   // nicht in Automatik
   #Mld.n_Auto := NOT #In.Auto AND "DB_ANLAGE".BA.Automat_ein;

   // Zeitüberschreitung links öffnen
   #IEC_Timer.TO_li_auf(IN := #Out.links_auf AND NOT #In.S_links_auf,
                        PT := #Param.TO,
                        Q => #TO_links_auf);
   IF #TO_links_auf THEN
       #Mld.TO_links_auf := TRUE;
   ELSIF #In.ErrQ THEN
       #Mld.TO_links_auf := FALSE;
   END_IF;
   // Zeitüberschreitung links schließen
   #IEC_Timer.TO_li_zu(IN := #Out.links_zu AND NOT #In.S_links_zu,
                        PT := #Param.TO,
                        Q => #TO_links_zu);
    IF #TO_links_zu THEN
        #Mld.TO_links_zu := TRUE;
    ELSIF #In.ErrQ THEN
        #Mld.TO_links_zu := FALSE;
    END_IF;
     // Zeitüberschreitung rechts öffnen
    #IEC_Timer.TO_re_auf(IN := #Out.rechts_auf AND NOT #In.S_rechts_auf,
                         PT := #Param.TO,
                         Q => #TO_rechts_auf);
    IF #TO_rechts_auf THEN
        #Mld.TO_rechts_auf := TRUE;
    ELSIF #In.ErrQ THEN
        #Mld.TO_rechts_auf := FALSE;
    END_IF;
    // Zeitüberschreitung rechts schließen
    #IEC_Timer.TO_re_zu(IN := #Out.rechts_zu AND NOT #In.S_rechts_zu,
                        PT := #Param.TO,
                        Q => #TO_rechts_zu);
    IF #TO_rechts_zu THEN
        #Mld.TO_rechts_zu := TRUE;
    ELSIF #In.ErrQ THEN
        #Mld.TO_rechts_zu := FALSE;
    END_IF;
   // Sensor und SRM Zylinder Zeitfenster überwachen 
    #IEC_Timer.gleich_li_auf(IN := #In.SRM_links_auf AND NOT #In.S_links_auf,
                             PT := #Param.gleichzeitig,
                             Q => #Mld.SF_gleich_li_auf);
    // Sensor und SRM Zylinder Zeitfenster überwachen 
    #IEC_Timer.gleich_li_zu(IN := #In.SRM_links_zu AND NOT #In.S_links_zu,
                             PT := #Param.gleichzeitig,
                             Q => #Mld.SF_gleich_li_zu);
     // Sensor und SRM Zylinder Zeitfenster überwachen 
     #IEC_Timer.gleich_re_auf(IN := #In.SRM_rechts_auf AND NOT #In.S_rechts_auf,
                             PT := #Param.gleichzeitig,
                             Q => #Mld.SF_gleich_re_auf);
    // Sensor und SRM Zylinder Zeitfenster überwachen 
    #IEC_Timer.gleich_re_zu(IN := #In.SRM_rechts_zu AND NOT #In.S_rechts_zu,
                            PT := #Param.gleichzeitig,
                            Q => #Mld.SF_gleich_re_zu);
END_REGION
END_FUNCTION_BLOCK

FUNCTION_BLOCK "RT"   // FB1192, LAD
TITLE = Torsteuerung
{ S7_Optimized_Access := 'TRUE' }
// stored: AutoNumber false, MemoryReserve 100, SetENOAutomatically true
   VAR RETAIN
      In { ExternalAccessible := 'False'; ExternalVisible := 'False'; ExternalWritable := 'False'} : Struct
         NotHalt : Bool;
         MSS_ok : Bool;
         ok : Bool;
         Knauf_Auto : Bool;
         T_auf : Bool;   // Paneltaste
         T_zu : Bool;   // Paneltaste
         S_auf : Bool;
         S_zu : Bool;
         ErrQ : Bool;   // Fehlerquittung
         Sperrluft_ok : Bool;
         Kein_Gas_Alarm : Bool;
      END_STRUCT;
      Param { ExternalAccessible := 'False'; ExternalVisible := 'False'; ExternalWritable := 'False'} : Struct
         "TO" : Time := T#3s500ms;
      END_STRUCT;
      Zst { ExternalAccessible := 'False'; ExternalVisible := 'False'; ExternalWritable := 'False'} : Struct
         Req_Auf : Bool;
         Fehler : Bool;
         Sperre_QF : Bool;
         QF_sicher : Bool;
      END_STRUCT;
      Out { ExternalAccessible := 'False'; ExternalVisible := 'False'; ExternalWritable := 'False'} : Struct
         auf : Bool;
         zu : Bool;
      END_STRUCT;
      Mld { ExternalAccessible := 'False'; ExternalVisible := 'False'; ExternalWritable := 'False'} : Struct
         n_Auto : Bool;
         TO_auf : Bool;
         TO_zu : Bool;
         MSS : Bool;
         nok : Bool;
      END_STRUCT;
   END_VAR
   VAR
      IEC_Timer { ExternalAccessible := 'False'; ExternalVisible := 'False'; ExternalWritable := 'False'} : Struct
         TO_auf : TON_TIME;
         TO_zu : TON_TIME;
      END_STRUCT;
   END_VAR
   VAR_TEMP
      TO_auf : Bool;
      TO_zu : Bool;
   END_VAR
BEGIN

REGION Network 1 (SCL): Input
   // Panelbdienung und Sensoren --> Input()
   // Not-Halt
   #In.NotHalt := NOT "DB_PNOZ_IN_Out".In.NH_Frg_RT;
   // kein Gasalarm
   #In.Kein_Gas_Alarm :="E_Al_Gas_ok";
   // Sperrluftventilator an
   #In.Sperrluft_ok := "A_Frg_FU_Vent";

   // Schnittstelle zum Transportsystem
   #Zst.QF_sicher :=("E_S_Pos_BE_QF1" OR "E_S_Pos_Ue_QF1") AND ("E_S_Pos_BE_QF2" OR "E_S_Pos_Ue_QF2")
   AND NOT "A_Frg_FU_QF_WR02" AND NOT "A_Frg_FU_QF_WR03";
END_REGION

REGION Network 2 (SCL): Sammelstörung
   IF #In.ErrQ THEN
       #Zst.Fehler := FALSE;
   END_IF;
   IF #In.NotHalt OR NOT #In.MSS_ok OR NOT #In.ok OR #Mld.TO_auf OR #Mld.TO_zu THEN
       #Zst.Fehler := TRUE;
   END_IF;
END_REGION

REGION Network 3 (SCL): Ansteuerung
   IF NOT #Zst.Fehler AND #In.Kein_Gas_Alarm AND #In.Sperrluft_ok THEN
       IF #In.Knauf_Auto THEN
           // Automatikbetrieb
           IF #Zst.QF_sicher THEN
               #Out.auf := #Zst.Req_Auf;// wird von WR02/03 gebildet
               #Out.zu := NOT #Zst.Req_Auf;
           ELSE
               #Out.auf := FALSE;
               #Out.zu := FALSE;
           END_IF;
       ELSE
           // Handbetrieb
           IF #In.T_auf AND NOT #In.T_zu THEN
               #Out.auf := TRUE;
               #Out.zu := FALSE;
           END_IF;
           IF #In.T_zu AND NOT #In.T_auf AND #Zst.QF_sicher THEN
               #Out.zu := TRUE;
               #Out.auf := FALSE;
           END_IF;
       END_IF;
   ELSE // Not-Halt, n.i.O, MSS
       #Out.auf := FALSE;
       #Out.zu := FALSE;
   END_IF;

   // Endlagen erreicht
   IF #In.S_auf THEN
       #Out.auf := FALSE;
   END_IF;

   IF #In.S_zu THEN
       #Out.zu := FALSE;
   END_IF;
END_REGION

REGION Network 4 (SCL): Sperre
   // Fahrt WR02/03  verboten
   #Zst.Sperre_QF := NOT #In.S_auf OR #In.S_zu OR #Out.zu;
END_REGION

REGION Network 5 (SCL): Überwachung / Alarme
   // MSS / Zeitüberschreitung
   // nicht betriebsbereit
   #Mld.nok := NOT #In.ok AND NOT #In.NotHalt;
   // Motorschutzschalter
   #Mld.MSS := NOT #In.MSS_ok AND NOT #In.NotHalt;

   // nicht in Automatik
   #Mld.n_Auto := NOT #In.Knauf_Auto AND "DB_ANLAGE".BA.Automat_ein;

   // Zeitüberschreitung öffnen
   #IEC_Timer.TO_auf(IN := #Out.auf AND NOT #In.S_auf,
                        PT := #Param.TO,
                        Q => #TO_auf);
      IF #TO_auf THEN
          #Mld.TO_auf := TRUE;
      ELSIF #In.ErrQ THEN
          #Mld.TO_auf := FALSE;
      END_IF;
          // Zeitüberschreitung schließen
   #IEC_Timer.TO_zu(IN := #Out.zu AND NOT #In.S_zu,
                        PT := #Param.TO,
                        Q => #TO_zu);
       IF #TO_zu THEN
           #Mld.TO_zu := TRUE;
       ELSIF #In.ErrQ THEN
           #Mld.TO_zu := FALSE;
       END_IF;
END_REGION
END_FUNCTION_BLOCK

FUNCTION_BLOCK "FP_Saeure.GP0x"   // FB1001, LAD
TITLE = Filterpumpe Säure
{ S7_Optimized_Access := 'TRUE' }
// Funktionen:  Filternn / /Filterwechsel / Spülen
// stored: AutoNumber false, MemoryReserve 100, SetENOAutomatically false
   VAR RETAIN
      In { ExternalAccessible := 'False'; ExternalVisible := 'False'; ExternalWritable := 'False'} : Struct
         NotHalt : Bool;
         ext_Freigabe : Bool;   // Kein Gasalarm, Kein Notstrom
         Auto : Bool;   // Paneltaste
         Ein : Bool;   // Paneltaste
         Quitt_FW : Bool;   // Paneltaste
         FU_betriebsbereit : Bool;
         FU_Stoerung : Bool;
         Niv_TLS : Bool;
         Niv_min : Bool;
         Niv_max : Bool;
         Niv_Uel : Bool;
         Frg_Niv_CM05 : Bool;
         Leckage_ok : Bool;
         SRM_Saugseite_auf : Bool;
         SRM_Saugseite_zu : Bool;
         SRM_Eingang_Filter_auf : Bool;
         SRM_Eingang_Filter_zu : Bool;
         SRM_Ausgang_Filter_auf : Bool;
         SRM_Ausgang_Filter_zu : Bool;
         SRM_Entluften_auf : Bool;
         SRM_Entlueften_zu : Bool;
         SRM_Eingang_Spülltg_P_auf : Bool;   // Pumpe
         SRM_Eingang_Spülltg_P_zu : Bool;   // Pumpe
         SRM_Eingang_Spülltg_F_auf : Bool;   // Filter
         SRM_Eingang_Spülltg_F_zu : Bool;   // Filter
         SRM_Ausgang_Spülltg_auf : Bool;
         SRM_Ausgang_Spülltg_zu : Bool;
         Sensor_FG_links : Bool;
         Sensor_FG_rechts : Bool;
         Einhausung_HQ0x_zu : Bool;
         GW_p_FP : Bool;
         GW_p_FG : Bool;
         GW_LF_FP : Bool;
         Betriebsart : USInt := 0;   // Paneltaste
         FU_speed : Int;
         Druck_Pumpe : Real;
         Delta_p_Filter : Real;
      END_STRUCT;
      Param { ExternalAccessible := 'False'; ExternalVisible := 'False'; ExternalWritable := 'False'} : Struct
         SW_Hand : Int;   // [%]
         SW_Auto_AZ : Int;   // [%]
         SW_Auto_aAZ : Int;   // [%]
         Spülzeit_Pumpe : Time;
         FG_Zeit_leeren_Saurebecken : Time;
         FG_Zeit_leeren_CM05 : Time;
         FW_Spülzeit : Time;
         FW_Wartezeit : Time;
         FW_Zeit_fuellen : Time;
         DT_Druckaufbau : Time;
         DT_Testzeit_Pumpe : Time;
         DT_Testzeit_Filter : Time;
         SW_Drucktest_Pumpe : Real;
         SW_Drucktest_Filter : Real;
         WarnGr_FW : Real;
         Wechsel_FW : Real;
         Name_Pumpe : String[12];
         Name_Filter : String[12];
      END_STRUCT;
      Zst { ExternalAccessible := 'False'; ExternalVisible := 'False'; ExternalWritable := 'False'} : Struct
         Status_GP0x : USInt;
         Status_FW : USInt;
         Status_DT_Pumpe : USInt;
         Status_DT_Filter : USInt;
         Restzeit_Spülen_Pumpe : Time;
         Restzeit_Filter : Time;
         Restzeit_DT : Time;
         Spuelen_Pumpe : Bool;
         Spuelen_Filter : Bool;
         Spuelen_aktiv : Bool;
         Drucktest_aktiv : Bool;
         Filtern : Bool;
         Zeit_laeuft : Bool;
         Drucktest_Pu_ok : Bool;
         Drucktest_Filter_ok : Bool;
         Bedienung_erlaubt : Bool;
         speed : Int;   // [%]
      END_STRUCT;
      Mld { ExternalAccessible := 'False'; ExternalVisible := 'False'; ExternalWritable := 'False'} : Struct
         Leckage : Bool;
         GW_p_FP : Bool;
         GW_LF_FP : Bool;
         GW_p_FG : Bool;
         FG_links_nicht_zu : Bool;
         FG_rechts_nicht_zu : Bool;
         Einhausung_nicht_zu : Bool;
         FU_nicht_bereit : Bool;
         FU_Stoerung : Bool;
         FG_Spülen_Ende : Bool;
         n_Auto : Bool;
         TO_Druckaufbau : Bool;
         Drucktest_Pumpe_ok : Bool;
         Drucktest_Pumpe_Fehler : Bool;
         Pu_Spuelen_Fertig : Bool;
         Drucktest_Filter_ok : Bool;
         Drucktest_Filter_Fehler : Bool;
         Drucktest_Filter_erfordert : Bool;
         Filterbeutel_Wechsel_Vorwarngrenze : Bool;
         Filterbeutel_Wechsel_notwendig : Bool;
      END_STRUCT;
      Out { ExternalAccessible := 'False'; ExternalVisible := 'False'; ExternalWritable := 'False'} : Struct
         GP0x_Ein : Bool;
         Ventil_Saugseite : Bool;
         Ventil_Eingang_Filter : Bool;
         Ventil_Ausgang_Filter : Bool;
         Ventil_Entlueften : Bool;
         Spülventil_P_Eingang : Bool;
         Spülventil_F_Eingang : Bool;
         Spülventil_Ausgang : Bool;
         Soll_speed : Int;
      END_STRUCT;
   END_VAR
   VAR
      IEC_Timer { ExternalAccessible := 'False'; ExternalVisible := 'False'; ExternalWritable := 'False'} : Struct
         Spülen_Pumpe { S7_SetPoint := 'True'} : TP_TIME;
         Filterwechsel { S7_SetPoint := 'True'} : TP_TIME;
         GW_p { S7_SetPoint := 'True'} : TON_TIME;
         Drucktest { S7_SetPoint := 'True'} : TP_TIME;
         TO_Druckaufbau { S7_SetPoint := 'True'} : TON_TIME;
         Verz_Ueberdruck { S7_SetPoint := 'True'} : TON_TIME;
         Spülventil_Ausgang { S7_SetPoint := 'True'} : TOF_TIME;
      END_STRUCT;
      R_TRIG_Hand_EIN { ExternalAccessible := 'False'; ExternalVisible := 'False'; ExternalWritable := 'False'} : R_TRIG;
   END_VAR
   VAR_TEMP
      Spülzeit_Pumpe : Time;
      Spülzeit_Filter : Time;
      Zeit_DT : Time;
      posFl_Hand : Bool;
      Filtergehäuse_ok : Bool;
   END_VAR
   VAR CONSTANT
      Niv_TLS : USInt := 2;
      Niv_Min : USInt := 20;
      Niv_max : USInt := 90;
      Niv_Uel : USInt := 98;
      S0 : USInt := 0;
      S1 : USInt := 1;
      S2 : USInt := 2;
      S3 : USInt := 3;
      S4 : USInt := 4;
      S5 : USInt := 5;
      S6 : USInt := 6;
      S7 : USInt := 7;
      S8 : USInt := 8;
      S10_FG_Leeren : USInt := 10;
   END_VAR
BEGIN

REGION Network 1 (SCL): Input
   // Panelbedienung und Sensoren --> Input()

    // positive Flanke "Hand Ein"
   #R_TRIG_Hand_EIN(CLK := #In.Ein,
                    Q => #posFl_Hand);
END_REGION

REGION Network 2 (SCL): Ansteuerung
   // Filtergehäuse geschlossen
   #Filtergehäuse_ok := #In.Sensor_FG_links AND #In.Sensor_FG_rechts AND #In.Einhausung_HQ0x_zu;

   // Alles AUS
   IF (#In.Betriebsart = 2) AND #In.Leckage_ok AND #In.ext_Freigabe THEN // Spülen
       // Ausschaltverzögert - Druckabbau
       #IEC_Timer.Spülventil_Ausgang(IN := #Out.Spülventil_P_Eingang,
                                     PT := T#3s,
                                     Q => #Out.Spülventil_Ausgang);
   ELSE
       #Out.Spülventil_P_Eingang := FALSE;
       #Out.Spülventil_Ausgang := FALSE;
   END_IF;
   #Out.Spülventil_F_Eingang := FALSE;
   #Zst.Restzeit_Spülen_Pumpe := T#0s;
   #Zst.Restzeit_Filter := T#0s;
   #Out.Ventil_Saugseite := FALSE;
   #Out.Ventil_Eingang_Filter := FALSE;
   #Out.Ventil_Entlueften := FALSE;
   #Out.Ventil_Ausgang_Filter := FALSE;

   // "Normal"-Betrieb
   #Zst.Bedienung_erlaubt := NOT #In.Ein AND NOT #In.Auto AND NOT #Mld.Drucktest_Pumpe_Fehler AND NOT #Mld.Drucktest_Filter_Fehler;

   //Drucktest Pumpe rücksetzen
   IF #In.Betriebsart <> 3 OR #Zst.Spuelen_aktiv OR #Zst.Filtern OR NOT #In.Ein THEN
       #Mld.Drucktest_Pumpe_ok := FALSE;
       // #Mld.Drucktest_Pumpe_Fehler := FALSE;
       #Zst.Status_DT_Pumpe := 0;
       #Zst.Drucktest_aktiv := FALSE;
   END_IF;
   //Drucktest Filter rücksetzen
   IF #In.Betriebsart <> 4 OR #Zst.Spuelen_aktiv OR #Zst.Filtern OR NOT #In.Ein THEN
       #Mld.Drucktest_Filter_ok := FALSE;
       // #Mld.Drucktest_Filter_Fehler := FALSE;
       #Zst.Status_DT_Filter := 0;
   END_IF;
   IF #In.Betriebsart <> 3 AND #In.Betriebsart <> 4 THEN
       #Mld.TO_Druckaufbau := FALSE;
   END_IF;
   //Filterwechsel rücksetzen
   IF #In.Betriebsart <> 1 OR #Zst.Spuelen_aktiv OR NOT #In.Ein THEN
       #Zst.Status_FW := 0;
   END_IF;
   //Spülmeldung rücksetzen
   IF #In.Betriebsart <> 2 OR NOT #In.Ein THEN
       #Mld.Pu_Spuelen_Fertig := FALSE;
   END_IF;
   IF #In.Leckage_ok AND #In.ext_Freigabe THEN
       CASE #In.Betriebsart OF
           0:  // Filterbetrieb
                         // Ventile öffnen
               IF NOT #Mld.Drucktest_Filter_erfordert AND NOT #Mld.Filterbeutel_Wechsel_notwendig THEN
                   #Out.Ventil_Saugseite := (#In.Auto OR #In.Ein) AND #In.Niv_TLS AND #In.SRM_Ausgang_Spülltg_zu AND #In.SRM_Eingang_Spülltg_P_zu AND #In.SRM_Eingang_Spülltg_F_zu;
                   #Out.Ventil_Eingang_Filter := #Out.Ventil_Saugseite;
                   #Out.Ventil_Ausgang_Filter := #Out.Ventil_Eingang_Filter;
               END_IF;
                   // Wenn geöffnet --> Frg Pumpe
                   #Zst.Filtern := #In.SRM_Eingang_Filter_auf AND #In.SRM_Ausgang_Filter_auf AND #In.SRM_Saugseite_auf;
                   // #Zst.Status_FW := #Ende;

           1:  // Filterwechsel 
               REGION Filterwechsel
                   #Zst.Filtern := FALSE;
                   CASE #Zst.Status_FW OF
                       #S0:  // Grundzustand
                           IF #In.Auto OR #In.Ein THEN
                               #Zst.Status_FW := #S1;
                           END_IF;

                       #S1:    // 1. Mal Leerlaufen ins Säurebecken - vor Spülen: Pumpe Aus - Ventile Auf - Zeit warten
                           // Ventile öffnen
                           #Out.Ventil_Eingang_Filter := #Filtergehäuse_ok AND #In.SRM_Ausgang_Spülltg_zu AND #In.SRM_Eingang_Spülltg_P_zu AND #In.SRM_Eingang_Spülltg_F_zu;
                           #Out.Ventil_Ausgang_Filter := #Out.Ventil_Eingang_Filter;
                           #Out.Ventil_Saugseite := #Out.Ventil_Eingang_Filter;
                           #Out.Ventil_Entlueften := #Out.Ventil_Eingang_Filter;

                           #IEC_Timer.Filterwechsel(IN := #In.SRM_Eingang_Filter_auf AND #In.SRM_Ausgang_Filter_auf AND #In.SRM_Saugseite_auf AND #In.SRM_Entluften_auf,
                                                    PT := #Param.FG_Zeit_leeren_Saurebecken,
                                                    ET => #Spülzeit_Filter,
                                                    Q => #Zst.Zeit_laeuft);
                           #Zst.Restzeit_Filter := #Param.FG_Zeit_leeren_Saurebecken - #Spülzeit_Filter;

                           IF NOT #Zst.Zeit_laeuft AND #In.SRM_Eingang_Filter_auf AND #In.SRM_Ausgang_Filter_auf AND #In.SRM_Saugseite_auf AND #In.SRM_Entluften_auf THEN
                               #Out.Ventil_Ausgang_Filter := #Out.Ventil_Eingang_Filter := #Out.Ventil_Saugseite := #Out.Ventil_Entlueften := FALSE;
                               #Zst.Status_FW := #S2;
                           END_IF;

                       #S2:    // Spülen Filtergehäuse
                           // Ventile öffnen
                           #Out.Spülventil_F_Eingang := #In.Frg_Niv_CM05;
                           #Out.Spülventil_Ausgang := NOT #Out.Ventil_Entlueften;
                           #Out.Ventil_Entlueften := #Zst.Zeit_laeuft AND #Zst.Restzeit_Filter < T#15s; //#Spülzeit_Filter > T#45s AND #Spülzeit_Filter <= T#60s;
                           #IEC_Timer.Filterwechsel(IN := #In.SRM_Ausgang_Spülltg_auf AND #In.SRM_Eingang_Spülltg_F_auf,
                                                    PT := #Param.FW_Spülzeit,
                                                    ET => #Spülzeit_Filter,
                                                    Q => #Zst.Zeit_laeuft);
                           #Zst.Restzeit_Filter := #Param.FW_Spülzeit - #Spülzeit_Filter;

                           IF NOT #Zst.Zeit_laeuft AND #In.SRM_Ausgang_Spülltg_auf AND #In.SRM_Eingang_Spülltg_F_auf THEN
                               #Out.Spülventil_F_Eingang := #Out.Spülventil_Ausgang := FALSE;
                               #Out.Ventil_Entlueften := FALSE;
                               #Zst.Status_FW := #S3;
                           END_IF;

                       #S3:    // Warten --> Meldung
                           #IEC_Timer.Filterwechsel(IN := #In.SRM_Ausgang_Spülltg_zu AND #In.SRM_Eingang_Spülltg_F_zu AND #In.SRM_Entlueften_zu,
                                                    PT := #Param.FW_Wartezeit,
                                                    ET => #Spülzeit_Filter,
                                                    Q => #Zst.Zeit_laeuft);
                           #Zst.Restzeit_Filter := #Param.FW_Wartezeit - #Spülzeit_Filter;
                           // Ventile öffnen
                           IF #Zst.Zeit_laeuft AND #Zst.Restzeit_Filter < t#10s THEN
                               #Out.Ventil_Entlueften := TRUE;// #Zst.Zeit_laeuft AND #Zst.Restzeit_Filter < t#10s; // #Spülzeit_Filter > T#45s AND #Spülzeit_Filter <= T#60s;
                               #Out.Spülventil_F_Eingang := #Out.Ventil_Entlueften;
                           ELSE
                               #Out.Ventil_Entlueften := FALSE;
                               #Out.Spülventil_F_Eingang := FALSE;
                           END_IF;

                           IF NOT #Zst.Zeit_laeuft AND #In.SRM_Eingang_Spülltg_F_auf AND #In.SRM_Entluften_auf THEN
                               #Zst.Status_FW := #S4;
                           END_IF;

                       #S4:    // 2. Mal Leerlaufen in CM05 - nach Spülen: Pumpe Aus - Ventile Auf - Zeit warten
                           // Ventile öffnen
                           #Out.Ventil_Saugseite := FALSE;
                         //  #Out.Ventil_Eingang_Filter := FALSE;  04.08.21
                           #Out.Spülventil_Ausgang :=  #In.Frg_Niv_CM05 (*AND #In.SRM_Ausgang_Filter_zu 04.08.21*) AND #In.SRM_Eingang_Spülltg_P_zu AND #In.SRM_Eingang_Spülltg_F_zu;
                           #Out.Ventil_Entlueften := #Out.Spülventil_Ausgang;

                           #IEC_Timer.Filterwechsel(IN :=  #In.Frg_Niv_CM05 (*AND #In.SRM_Eingang_Filter_zu 04.08.21*) AND #In.SRM_Ausgang_Spülltg_auf AND #In.SRM_Saugseite_zu AND #In.SRM_Entluften_auf,
                                                    PT := #Param.FG_Zeit_leeren_CM05,
                                                    ET => #Spülzeit_Filter,
                                                    Q => #Zst.Zeit_laeuft);
                           #Zst.Restzeit_Filter := #Param.FG_Zeit_leeren_CM05 - #Spülzeit_Filter;

                           // 03.08.21
                           //Eine Bitte habe ich noch, zwar beim Filterwechsel. Es steht immer noch recht viel restliches saures Wasser im Behälter,
                           //könntest du bitte für den letzten Schritt noch 10sec für HQ01 den QM23 und bei HQ02 den QM60 öffnen.
                           //Somit ist auch die Leitung zur Leitfähigkeitsmessung leer.
                           #Out.Ventil_Eingang_Filter := #Out.Ventil_Ausgang_Filter := #Zst.Zeit_laeuft AND #Zst.Restzeit_Filter <= t#40s;// 03.08.21

                           IF NOT #Zst.Zeit_laeuft (*AND #In.SRM_Eingang_Filter_zu 04.08.21*) AND #In.SRM_Ausgang_Spülltg_auf AND #In.SRM_Saugseite_zu AND #In.SRM_Entluften_auf THEN
                               #Out.Ventil_Ausgang_Filter := #Out.Ventil_Eingang_Filter := #Out.Ventil_Saugseite := #Out.Ventil_Entlueften := FALSE;
                               #Zst.Status_FW := #S5;
                               #Mld.FG_Spülen_Ende := TRUE;
                           END_IF;

                       #S5:    // man.Wechsel --> Quittierung
                           // Ventile bleiben offen --> Nachlauf Restwasser in CM05
                           #Out.Ventil_Saugseite := FALSE;
                           #Out.Ventil_Eingang_Filter := FALSE;
                           #Out.Spülventil_Ausgang := #In.Frg_Niv_CM05 AND #In.SRM_Ausgang_Filter_zu AND #In.SRM_Eingang_Spülltg_P_zu AND #In.SRM_Eingang_Spülltg_F_zu;
                           #Out.Ventil_Entlueften := #Out.Spülventil_Ausgang;

                           IF #Filtergehäuse_ok AND #In.Quitt_FW THEN
                               #Mld.FG_Spülen_Ende := FALSE;
                               #Mld.Drucktest_Filter_erfordert := TRUE;
                               #Mld.Filterbeutel_Wechsel_notwendig := FALSE;
                               #In.Quitt_FW := FALSE;
                               #Zst.Status_FW := #S8;
                           END_IF;

                           (*     
                            #S6:    //Filtergehäuse füllen
                                #Out.Ventil_Saugseite := (#In.Auto OR #In.Ein) AND #In.Niv_TLS AND #In.SRM_Ausgang_Spülltg_zu AND #In.SRM_Eingang_Spülltg_P_zu AND #In.SRM_Eingang_Spülltg_F_zu;
                                #Out.Ventil_Eingang_Filter := #Out.Ventil_Saugseite;
                                #Out.Ventil_Ausgang_Filter := TRUE;
                                #Out.Spülventil_Ausgang := FALSE;

                                // Wenn geöffnet --> Frg Pumpe
                                #IEC_Timer.Filterwechsel(IN := #In.SRM_Eingang_Filter_auf AND #In.SRM_Saugseite_auf AND #In.SRM_Ausgang_Filter_auf,
                                                         PT := #Param.FW_Zeit_fuellen,
                                                         ET => #Spülzeit_Filter,
                                                         Q => #Zst.Zeit_laeuft);

                                #Zst.Filtern := #In.SRM_Eingang_Filter_auf AND #In.SRM_Ausgang_Filter_auf AND #In.SRM_Saugseite_auf;

                                #Zst.Restzeit_Filter := #Param.FW_Zeit_fuellen - #Spülzeit_Filter;

                                IF NOT #Zst.Zeit_laeuft AND #Zst.Filtern THEN
                                    #Zst.Status_FW := #S7;
                                END_IF;


                            #S7:    // Kreislauf öffnen
                                // #Out.Ventil_Ausgang_Filter := TRUE;
                                // #Out.Spülventil_Ausgang := NOT #In.SRM_Ausgang_Filter_auf;

                                // IF #In.SRM_Ausgang_Filter_auf AND #In.SRM_Ausgang_Spülltg_zu THEN
                                //     #Zst.Status_FW := #S8;
                                // END_IF;
                                #Zst.Filtern := FALSE;
                                IF #Zst.speed <= 20 THEN
                                    #Out.Ventil_Saugseite := FALSE;
                                    #Out.Ventil_Eingang_Filter := FALSE;
                                    #Out.Ventil_Ausgang_Filter := FALSE;
                                    #Out.Spülventil_Ausgang := FALSE;
                                END_IF;

                                IF NOT  #Zst.Filtern AND  #In.SRM_Saugseite_zu AND #In.SRM_Eingang_Filter_zu AND #In.SRM_Ausgang_Filter_zu AND #In.SRM_Ausgang_Spülltg_zu THEN
                                    #Zst.Status_FW := #S8;
                                END_IF;
                                  *)
                       #S8: // Ende
                           ;
                   END_CASE;
               END_REGION

           2:// Spülen - nur Hand
               #Zst.Filtern := FALSE;
               #Zst.Status_FW := #S0;

               IF NOT #Mld.Drucktest_Filter_erfordert AND NOT #Mld.Filterbeutel_Wechsel_notwendig THEN
                   IF #In.Ein AND #In.Frg_Niv_CM05 THEN
                       IF #posFl_Hand THEN
                           #Zst.Spuelen_aktiv := TRUE;
                       END_IF;
                       #Out.Spülventil_P_Eingang := #Filtergehäuse_ok AND #In.SRM_Ausgang_Filter_zu AND #In.SRM_Saugseite_zu AND #Zst.Spuelen_aktiv;
                       #Out.Ventil_Eingang_Filter := #Out.Spülventil_Ausgang;

                       #IEC_Timer.Spülen_Pumpe(IN := #In.SRM_Eingang_Spülltg_P_auf AND #In.SRM_Ausgang_Spülltg_auf,
                                               PT := #Param.Spülzeit_Pumpe,
                                               Q => #Zst.Spuelen_Pumpe,
                                               ET => #Spülzeit_Pumpe);
                       #Zst.Restzeit_Spülen_Pumpe := #Param.Spülzeit_Pumpe - #Spülzeit_Pumpe;

                       IF #In.SRM_Eingang_Spülltg_P_auf AND #In.SRM_Ausgang_Spülltg_auf AND NOT #Zst.Spuelen_Pumpe THEN
                           #Zst.Spuelen_aktiv := FALSE;
                           #Out.Spülventil_P_Eingang := FALSE;
                       END_IF;

                       // Fertig
                       IF NOT #Zst.Spuelen_Pumpe AND NOT #Zst.Spuelen_aktiv AND NOT #Out.Spülventil_Ausgang THEN
                           #Out.Spülventil_P_Eingang := FALSE;
                           #Out.Spülventil_Ausgang := FALSE;
                           #Out.Ventil_Eingang_Filter := FALSE;
                           #Zst.Restzeit_Spülen_Pumpe := T#0s;
                           #Mld.Pu_Spuelen_Fertig := TRUE;
                       END_IF;
                   ELSE
                       #Zst.Spuelen_Pumpe := FALSE;
                       #Out.Spülventil_P_Eingang := FALSE;
                       #Out.Spülventil_Ausgang := FALSE;
                       #Out.Ventil_Eingang_Filter := FALSE;
                       #Zst.Restzeit_Spülen_Pumpe := T#0s;
                   END_IF;
                   // Ausschaltverzögert - Druckabbau
                   #IEC_Timer.Spülventil_Ausgang(IN := #Out.Spülventil_P_Eingang,
                                                 PT := T#3s,
                                                 Q => #Out.Spülventil_Ausgang);
               END_IF;
           3: // Spülen + Drucktest - nur Hand
               #Zst.Filtern := FALSE;
               #Zst.Status_FW := #S0;
               IF NOT #Mld.Drucktest_Filter_erfordert AND NOT #Mld.Filterbeutel_Wechsel_notwendig THEN
                   IF NOT #Zst.Drucktest_aktiv THEN
                       IF #In.Ein AND #In.Frg_Niv_CM05 THEN
                           IF #posFl_Hand THEN
                               #Zst.Spuelen_aktiv := TRUE;
                           END_IF;
                           #Out.Spülventil_P_Eingang := #Filtergehäuse_ok AND #In.SRM_Ausgang_Filter_zu AND #In.SRM_Saugseite_zu;
                           #Out.Spülventil_Ausgang := #Out.Spülventil_P_Eingang;
                           #Out.Ventil_Eingang_Filter := #Out.Spülventil_P_Eingang;

                           #IEC_Timer.Spülen_Pumpe(IN := #In.SRM_Eingang_Spülltg_P_auf AND #In.SRM_Ausgang_Spülltg_auf,
                                                   PT := #Param.Spülzeit_Pumpe,
                                                   Q => #Zst.Spuelen_Pumpe,
                                                   ET => #Spülzeit_Pumpe);
                           #Zst.Restzeit_Spülen_Pumpe := #Param.Spülzeit_Pumpe - #Spülzeit_Pumpe;

                           IF #In.SRM_Eingang_Spülltg_P_auf AND #In.SRM_Ausgang_Spülltg_auf AND NOT #Zst.Spuelen_Pumpe THEN
                               #Zst.Spuelen_aktiv := FALSE;
                           END_IF;

                           // Fertig
                           IF NOT #Zst.Spuelen_Pumpe AND NOT #Zst.Spuelen_aktiv THEN
                               #Out.Spülventil_Ausgang := FALSE;
                               #Out.Ventil_Eingang_Filter := FALSE;
                               #Zst.Restzeit_Spülen_Pumpe := T#0s;
                               #Zst.Drucktest_aktiv := TRUE;
                               #Zst.Status_DT_Pumpe := #S1;
                           END_IF;
                       ELSE
                           #Zst.Spuelen_Pumpe := FALSE;
                           #Out.Spülventil_P_Eingang := FALSE;
                           #Out.Spülventil_Ausgang := FALSE;
                           #Out.Ventil_Eingang_Filter := FALSE;
                           #Zst.Restzeit_Spülen_Pumpe := T#0s;
                       END_IF;
                   END_IF;


                   //Drucktest
                   IF #Zst.Drucktest_aktiv THEN

                       CASE #Zst.Status_DT_Pumpe OF
                           #S1:  //Druckaufbau

                               IF "DB_Temporaer".Drucksensoren_deaktiviert THEN //20.01.22
                                   #Zst.Drucktest_Pu_ok := TRUE;

                                   "Ergebnis_DT"("Name" := #Param.Name_Pumpe,
                                                 akt_Zeit := "Uhrzeit".aktDatum,
                                                 ok := #Zst.Drucktest_Pu_ok,
                                                 Fehler := NOT #Zst.Drucktest_Pu_ok);

                                   #Mld.Drucktest_Pumpe_ok := #Zst.Drucktest_Pu_ok;
                                   #Mld.Drucktest_Pumpe_Fehler := NOT #Zst.Drucktest_Pu_ok;

                                   #Zst.Status_DT_Pumpe := #S4;
                               ELSE
                                   #Out.Spülventil_P_Eingang := #In.SRM_Ausgang_Filter_zu AND #In.SRM_Saugseite_zu;
                                   #Out.Ventil_Eingang_Filter := FALSE;
                                   #Out.Spülventil_Ausgang := FALSE;

                                   IF (#In.Druck_Pumpe > #Param.SW_Drucktest_Pumpe + 0.25 AND #In.SRM_Eingang_Filter_zu) OR #Mld.TO_Druckaufbau THEN
                                       #Out.Spülventil_P_Eingang := FALSE;
                                       #Zst.Status_DT_Pumpe := #S2;
                                   END_IF;

                               END_IF;

                           #S2: //Wartezeit
                               #IEC_Timer.Drucktest(IN := #In.SRM_Eingang_Spülltg_P_zu,
                                                    PT := #Param.DT_Testzeit_Pumpe,
                                                    Q => #Zst.Zeit_laeuft,
                                                    ET => #Zeit_DT);
                               #Zst.Restzeit_DT := #Param.DT_Testzeit_Pumpe - #Zeit_DT;

                               IF NOT #Zst.Zeit_laeuft AND #In.SRM_Eingang_Spülltg_P_zu THEN
                                   #Zst.Restzeit_DT := T#0s;
                                   #Zst.Status_DT_Pumpe := #S3;
                               END_IF;

                           #S3:// Überprüfung
                               #Zst.Drucktest_Pu_ok := #In.Druck_Pumpe >= #Param.SW_Drucktest_Pumpe;

                               "Ergebnis_DT"("Name" := #Param.Name_Pumpe,
                                             akt_Zeit := "Uhrzeit".aktDatum,
                                             ok := #Zst.Drucktest_Pu_ok,
                                             Fehler := NOT #Zst.Drucktest_Pu_ok);

                               #Mld.Drucktest_Pumpe_ok := #Zst.Drucktest_Pu_ok;
                               #Mld.Drucktest_Pumpe_Fehler := NOT #Zst.Drucktest_Pu_ok;

                               #Zst.Status_DT_Pumpe := #S4;

                           #S4: // ENDE
                               ;
                       END_CASE;
                   END_IF;
               END_IF;
           4: // Drucktest Filter
               #Zst.Filtern := FALSE;
               IF #posFl_Hand (*AND NOT #Mld.Filterbeutel_Wechsel_notwendig - 23.08.22, falls während Drucktest die Meldung aktiv wird, dass es nicht im deadlock ist*) THEN
                   #Zst.Status_DT_Filter:= 1;
               END_IF;

               CASE #Zst.Status_DT_Filter OF
                   #S1:  //Druckaufbau

                       IF "DB_Temporaer".Drucksensoren_deaktiviert THEN //20.01.22
                           #Zst.Drucktest_Filter_ok := TRUE;

                           "Ergebnis_DT"("Name" := #Param.Name_Filter,
                                         akt_Zeit := "Uhrzeit".aktDatum,
                                         ok := #Zst.Drucktest_Filter_ok,
                                         Fehler := NOT #Zst.Drucktest_Filter_ok);

                           #Mld.Drucktest_Filter_ok := #Zst.Drucktest_Filter_ok;
                           #Mld.Drucktest_Filter_Fehler := NOT #Zst.Drucktest_Filter_ok;
                           #Mld.Drucktest_Filter_erfordert := FALSE;
                           #Zst.Status_DT_Filter := #S10_FG_Leeren;

                       ELSE
                           #Out.Spülventil_F_Eingang := #Filtergehäuse_ok AND #In.SRM_Ausgang_Filter_zu AND #In.SRM_Saugseite_zu;
                           #Out.Ventil_Eingang_Filter := FALSE;
                           #Out.Spülventil_Ausgang := FALSE;

                           IF (ABS(#In.Delta_p_Filter) > #Param.SW_Drucktest_Filter + 0.25 AND #In.SRM_Eingang_Spülltg_F_auf) OR #Mld.TO_Druckaufbau OR #Mld.GW_p_FG THEN
                               #Out.Spülventil_F_Eingang := FALSE;
                               #Zst.Status_DT_Filter := #S2;
                           END_IF;
                           #Zst.Restzeit_DT := #Param.DT_Druckaufbau - #IEC_Timer.TO_Druckaufbau.ET;

                       END_IF;

                   #S2: //Wartezeit
                       #IEC_Timer.Drucktest(IN := #In.SRM_Eingang_Spülltg_F_zu,
                                            PT := #Param.DT_Testzeit_Filter,
                                            Q => #Zst.Zeit_laeuft,
                                            ET => #Zeit_DT);
                       #Zst.Restzeit_DT := #Param.DT_Testzeit_Filter - #Zeit_DT;

                       IF NOT #Zst.Zeit_laeuft AND #In.SRM_Eingang_Spülltg_F_zu THEN
                           #Zst.Restzeit_DT := T#0s;
                           #Zst.Status_DT_Filter := #S3;
                       END_IF;

                   #S3:// Überprüfung
                       #Zst.Drucktest_Filter_ok := ABS(#In.Delta_p_Filter) >= #Param.SW_Drucktest_Filter;

                       "Ergebnis_DT"("Name" := #Param.Name_Filter,
                                     akt_Zeit := "Uhrzeit".aktDatum,
                                     ok := #Zst.Drucktest_Filter_ok,
                                     Fehler := NOT #Zst.Drucktest_Filter_ok);

                       #Mld.Drucktest_Filter_ok := #Zst.Drucktest_Filter_ok;
                       #Mld.Drucktest_Filter_Fehler := NOT #Zst.Drucktest_Filter_ok;
                       #Mld.Drucktest_Filter_erfordert := FALSE;
                       #Zst.Status_DT_Filter := #S10_FG_Leeren;

                   #S10_FG_Leeren: // Filtergehäuse nach NIO Drucktest leeren in CM05
                       // Ventile öffnen
                       #Out.Ventil_Saugseite := FALSE;
                     //#Out.Ventil_Eingang_Filter := FALSE;  04.08.21
                       #Out.Spülventil_Ausgang := #In.Frg_Niv_CM05 (*AND #In.SRM_Ausgang_Filter_zu 04.08.21*) AND #In.SRM_Eingang_Spülltg_P_zu AND #In.SRM_Eingang_Spülltg_F_zu;;
                       #Out.Ventil_Entlueften :=  #Out.Spülventil_Ausgang;

                       #IEC_Timer.Filterwechsel(IN := #In.Frg_Niv_CM05 (*AND #In.SRM_Eingang_Filter_zu04.08.21*)AND #In.SRM_Ausgang_Spülltg_auf AND #In.SRM_Saugseite_zu AND #In.SRM_Entluften_auf,
                                                PT := #Param.FG_Zeit_leeren_CM05,
                                                ET => #Spülzeit_Filter,
                                                Q => #Zst.Zeit_laeuft);
                       #Zst.Restzeit_DT := #Param.FG_Zeit_leeren_CM05 - #Spülzeit_Filter;

                       // 04.08.21
                       //Eine Bitte habe ich noch, zwar beim Filterwechsel. Es steht immer noch recht viel restliches saures Wasser im Behälter,
                       //könntest du bitte für den letzten Schritt noch 10sec für HQ01 den QM23 und bei HQ02 den QM60 öffnen.
                       //Somit ist auch die Leitung zur Leitfähigkeitsmessung leer.
                       #Out.Ventil_Eingang_Filter := #Out.Ventil_Ausgang_Filter := #Zst.Zeit_laeuft AND #Zst.Restzeit_DT <= t#40s;// 03.08.21

                       IF NOT #Zst.Zeit_laeuft (*AND #In.SRM_Eingang_Filter_zu04.08.21*)AND #In.SRM_Ausgang_Spülltg_auf AND #In.SRM_Saugseite_zu AND #In.SRM_Entluften_auf THEN
                           #Out.Spülventil_Ausgang := #Out.Ventil_Eingang_Filter := #Out.Ventil_Saugseite := #Out.Ventil_Entlueften := FALSE;
                           #Zst.Status_DT_Filter := #S4;
                       END_IF;

                   #S4: // ENDE
                       ;


               END_CASE;

       END_CASE;
   END_IF;

       // Pumpe an    
   #Out.GP0x_Ein := #Zst.Filtern AND NOT #In.NotHalt AND #Filtergehäuse_ok AND #In.Leckage_ok AND #In.ext_Freigabe AND (#In.Ein OR #In.Auto);

       // Geschwindigkeitsvorgabe
       // SEW: 100% == 3000 U/min == 15000 Digits
       IF #Out.GP0x_Ein THEN
           IF #In.Ein THEN
               #Out.Soll_speed := #Param.SW_Hand * 150;
           ELSE
               IF "Uhrzeit".AZ_aktiv THEN
                   #Out.Soll_speed := #Param.SW_Auto_AZ * 150;
               ELSE
                   #Out.Soll_speed := #Param.SW_Auto_aAZ * 150;
               END_IF;
           END_IF;
       ELSE
           #Out.Soll_speed := 0;
       END_IF;
END_REGION

REGION Network 3 (SCL): Überwachung / Meldungen
   // Leckage
   #Mld.Leckage := NOT #In.Leckage_ok;

   // Zeitüberschreitung Druckaufbau
   #IEC_Timer.TO_Druckaufbau(IN := #Zst.Status_DT_Pumpe = #S1 OR #Zst.Status_DT_Filter = #S1,
                             PT := #Param.DT_Druckaufbau,
                             Q => #Mld.TO_Druckaufbau);

   //Grenzwert Druck Filtergehäuse
   #IEC_Timer.Verz_Ueberdruck(IN := #In.GW_p_FG,
                              PT :=t#3s,
                              Q => #Mld.GW_p_FG);

   // Nicht geschlossen
   #Mld.Einhausung_nicht_zu := NOT #In.Einhausung_HQ0x_zu;
   #Mld.FG_links_nicht_zu := NOT #In.Sensor_FG_links;
   #Mld.FG_rechts_nicht_zu := NOT #In.Sensor_FG_rechts;

   // Grenzwert Druck Pumpe
   #IEC_Timer.GW_p(IN :=#Out.GP0x_Ein AND #In.GW_p_FP,
                   PT := T#3s,
                   Q => #Mld.GW_p_FP);
   // Grenzwert Leitfähigkeit
   #Mld.GW_LF_FP := #In.GW_LF_FP;

   // Frequenzumrichter 24V-Betrieb
   #Mld.FU_nicht_bereit := NOT #In.FU_betriebsbereit AND NOT #In.NotHalt;
   // Störung Frequenzumrichter
   #Mld.FU_Stoerung := #In.FU_Stoerung AND NOT #In.NotHalt;
   // nicht in Automatik
   #Mld.n_Auto := NOT #In.Auto AND "DB_ANLAGE".BA.Automat_ein;
   // Filterwechsel
   #Mld.Filterbeutel_Wechsel_Vorwarngrenze := #In.Delta_p_Filter > #Param.WarnGr_FW AND NOT #Mld.Filterbeutel_Wechsel_notwendig;

   IF #In.Delta_p_Filter > #Param.Wechsel_FW THEN
       #Mld.Filterbeutel_Wechsel_notwendig := TRUE;
   END_IF;
END_REGION

REGION Network 4 (SCL): --> Visu
   // Status Pumpe
   "Status_E0A"(Hand := #In.Ein,
                Auto := #In.Auto,
                SonderModus_PumpeSpuelen:=#Zst.Spuelen_Pumpe,
                Stoerung := #In.FU_Stoerung OR NOT #In.FU_betriebsbereit,
                Ausgang := #Out.GP0x_Ein,
                StatusByte => #Zst.Status_GP0x);

   // Ist-Geschwindigkeit FU
   // SEW: 100% == 3000 U/min == 15000 Digits
   #Zst.speed := #In.FU_speed / 150; // in[%]
END_REGION
END_FUNCTION_BLOCK

FUNCTION_BLOCK "UP_Saeure.GP0x"   // FB1002, LAD
TITLE = Pumpe Umwälzpumpe Säure
{ S7_Optimized_Access := 'TRUE' }
// Funktionen: Umwälzen / Entsorgung
// stored: AutoNumber false, MemoryReserve 100, SetENOAutomatically false
   VAR RETAIN
      In { ExternalAccessible := 'False'; ExternalVisible := 'False'; ExternalWritable := 'False'} : Struct
         NotHalt : Bool;
         ext_Freigabe : Bool;   // Kein Gasalarm, Kein Notstrom
         TW_senkt : Bool;
         Auto : Bool;   // Paneltaste
         Ein : Bool;   // Paneltaste
         Quitt_Al_Dfl : Bool;
         FU_betriebsbereit : Bool;
         FU_Stoerung : Bool;
         Niv_TLS : Bool;
         Niv_min : Bool;
         Niv_max : Bool;
         Niv_Uel : Bool;
         Frg_Niv_CM05 : Bool;
         SRM_Saugseite_auf : Bool;
         SRM_Saugseite_zu : Bool;
         SRM_Druckseite_auf : Bool;
         SRM_Druckseite_zu : Bool;
         SRM_Eingang_Spülltg_auf : Bool;
         SRM_Eingang_Spülltg_zu : Bool;
         SRM_Ausgang_Spülltg_auf : Bool;
         SRM_Ausgang_Spülltg_zu : Bool;
         SRM_Entsogung_UV02_auf : Bool;
         SRM_Entsogung_UV02_zu : Bool;
         SRM_UV02_GP01_auf : Bool;
         SRM_UV02_GP01_zu : Bool;
         SRM_UV02_GP02_auf : Bool;
         SRM_UV02_GP02_zu : Bool;
         "SRM_GP02.QM41_auf" : Bool;
         "SRM_GP01.QM14_auf" : Bool;
         Anf_HF_Ents_CM0x : Bool;
         GW_p_UP : Bool;
         GW_LF_UP : Bool;
         Imp_Dfl : Bool;
         GW_Dfl : Bool;
         Tuer_zu_Seite_GP01 : Bool;
         Tuer_zu_vorn_GP01 : Bool;
         Tuer_zu_vorn_GP02 : Bool;
         Leckage_Doppelrohr_ok_BL26 : Bool;
         Leckage_Doppelschlauch_ok_BL33 : Bool;
         Leckage_Uml_Tunnel_ok_BL34 : Bool;
         Leckage_PFA_Uebergang_ok_BL16 : Bool;
         Leckage_PFA_Uebergang_ok_BL25 : Bool;
         Betriebsart : USInt := 0;   // Paneltaste
         FU_speed : Int;
         Druck_Pumpe : Real;
      END_STRUCT;
      Param { ExternalAccessible := 'False'; ExternalVisible := 'False'; ExternalWritable := 'False'} : Struct
         SW_Hand : Int;   // [%]
         SW_Auto_AZ : Int;   // [%]
         SW_Auto_aAZ : Int;   // [%]
         Spülzeit : Time;
         DT_Druckaufbau : Time;
         DT_Testzeit : Time;
         SW_Drucktest : Real;
         "Name" : String[12];
      END_STRUCT;
      Zst { ExternalAccessible := 'False'; ExternalVisible := 'False'; ExternalWritable := 'False'} : Struct
         Niveau : USInt;
         Status_GP0x : USInt;
         Status_DT : USInt;
         Restzeit_Spülen : Time;
         Restzeit_DT : Time;
         Spuelen : Bool;
         Spuelen_aktiv : Bool;
         Drucktest_aktiv : Bool;
         Umwaelzen : Bool;
         Weg_frei : Bool;
         Zeit_laeuft : Bool;
         Drucktest_ok : Bool;
         Bedienung_erlaubt : Bool;
         speed : Int;   // [%]
      END_STRUCT;
      Mld { ExternalAccessible := 'False'; ExternalVisible := 'False'; ExternalWritable := 'False'} : Struct
         Niv_TLS : Bool;
         Niv_Ueberlauf : Bool;
         Niv_Sensorfehler : Bool;
         GW_p_UP : Bool;
         GW_LF_UP : Bool;
         GW_Dfl : Bool;
         UeW_Dfl_Ents : Bool;
         FU_nicht_bereit : Bool;
         FU_Stoerung : Bool;
         n_Auto : Bool;
         TO_Druckaufbau : Bool;
         Drucktest_ok : Bool;
         DT_Fehler : Bool;
         Pu_Spuelen_Fertig : Bool;
      END_STRUCT;
      Out { ExternalAccessible := 'False'; ExternalVisible := 'False'; ExternalWritable := 'False'} : Struct
         GP0x_Ein : Bool;
         Ventil_Saugseite : Bool;
         Ventil_Druckseite : Bool;
         Spülventil_Eingang : Bool;
         Spülventil_Ausgang : Bool;
         Entsorgung_UV02 : Bool;
         Ventil_UV02_GP01 : Bool;
         Ventil_UV02_GP02 : Bool;
         Soll_speed : Int;
      END_STRUCT;
   END_VAR
   VAR
      IEC_Timer { ExternalAccessible := 'False'; ExternalVisible := 'False'; ExternalWritable := 'False'} : Struct
         Spülen { S7_SetPoint := 'True'} : TP_TIME;
         GW_p { S7_SetPoint := 'True'} : TON_TIME;
         GW_Dfl { S7_SetPoint := 'True'} : TON_TIME;
         Imp_Dfl { S7_SetPoint := 'True'} : TON_TIME;
         Drucktest { S7_SetPoint := 'True'} : TP_TIME;
         TO_Druckaufbau { S7_SetPoint := 'True'} : TON_TIME;
         Spülventil_Ausgang { S7_SetPoint := 'True'} : TOF_TIME;
      END_STRUCT;
      R_TRIG_Hand_EIN { ExternalAccessible := 'False'; ExternalVisible := 'False'; ExternalWritable := 'False'} : R_TRIG;
   END_VAR
   VAR_TEMP
      Spülzeit : Time;
      Zeit_DT : Time;
      posFl_Hand : Bool;
      Leckage_Entsorgung_ok_GP01 : Bool;
      Leckage_Entsorgung_ok_GP02 : Bool;
      Alarm_Dfl_Ents : Bool;
   END_VAR
   VAR CONSTANT
      Niv_TLS : USInt := 7;
      Niv_Min : USInt := 70;
      Niv_max : USInt := 85;
      Niv_Uel : USInt := 98;
      S1 : USInt := 1;
      S2 : USInt := 2;
      S3 : USInt := 3;
      S4 : USInt := 4;
   END_VAR
BEGIN

REGION Network 1 (SCL): Input
   // Panelbedienung und Sensoren --> Input()
   // Not-Halt
   #In.NotHalt := NOT "DB_PNOZ_IN_Out".In.NH_Frg_Pumpen OR NOT "E_Frg_AbLW";

    // positive Flanke "Hand Ein"
   #R_TRIG_Hand_EIN(CLK := #In.Ein,
                    Q => #posFl_Hand);

   // Leckage Entsorgung
   #Leckage_Entsorgung_ok_GP01 :=#In.Leckage_PFA_Uebergang_ok_BL16 AND #In.Leckage_Doppelrohr_ok_BL26 AND #In.Leckage_Uml_Tunnel_ok_BL34;

   #Leckage_Entsorgung_ok_GP02 := #In.Leckage_PFA_Uebergang_ok_BL25 AND #In.Leckage_Doppelrohr_ok_BL26 AND #In.Leckage_Doppelschlauch_ok_BL33;

   // Quittierung Alarm Durchfluss
   IF #In.Quitt_Al_Dfl AND #Mld.UeW_Dfl_Ents THEN
       #Mld.UeW_Dfl_Ents := FALSE;
   END_IF;
END_REGION

REGION Network 2 (SCL): Ansteuerung
   // Alles AUS
   IF (#In.Betriebsart = 3) AND #In.ext_Freigabe THEN // Spülen
       #IEC_Timer.Spülventil_Ausgang(IN := #Out.Spülventil_Eingang,
                                     PT := T#3s,
                                     Q => #Out.Spülventil_Ausgang);
   ELSE
       #Out.Spülventil_Eingang := FALSE;
       #Out.Spülventil_Ausgang := FALSE;
   END_IF;
   #Zst.Restzeit_Spülen := T#0s;
   #Out.Ventil_Saugseite := FALSE;
   #Out.Ventil_Druckseite := FALSE;
   #Out.Entsorgung_UV02 := FALSE;
   #Out.Ventil_UV02_GP01 := FALSE;
   #Out.Ventil_UV02_GP02 := FALSE;

   // "Normal"-Betrieb
   #Zst.Bedienung_erlaubt := NOT #In.Ein AND NOT #In.Auto AND NOT #Mld.DT_Fehler;

   //Drucktest rücksetzen
   IF #In.Betriebsart <> 4 OR #Zst.Spuelen_aktiv OR #Zst.Umwaelzen OR NOT #In.Ein THEN
       #Mld.Drucktest_ok := FALSE;
       // #Mld.DT_Fehler := FALSE;
       #Mld.TO_Druckaufbau := FALSE;
       #Zst.Status_DT := 0;
       #Zst.Drucktest_aktiv := FALSE;
   END_IF;
   //Spülmeldung rücksetzen
   IF #In.Betriebsart <> 3 OR NOT #In.Ein THEN
       #Mld.Pu_Spuelen_Fertig := FALSE;
   END_IF;

   IF #In.ext_Freigabe THEN
       CASE #In.Betriebsart OF
           0:  // Umwälzen
                     // Ventile öffnen
               #Out.Ventil_Saugseite := (#In.Auto OR #In.Ein) AND #In.Niv_TLS AND NOT #In.TW_senkt
               AND #In.SRM_Ausgang_Spülltg_zu AND #In.SRM_Eingang_Spülltg_zu;
               #Out.Ventil_Druckseite := #Out.Ventil_Saugseite AND NOT #In.Anf_HF_Ents_CM0x;

               // Verwerfen Auto
               #Out.Ventil_UV02_GP01 := #In.Anf_HF_Ents_CM0x AND #In."SRM_GP01.QM14_auf" AND #In.Auto
               AND #In.Tuer_zu_Seite_GP01 AND #In.Tuer_zu_vorn_GP01 AND #Leckage_Entsorgung_ok_GP01;

               #Out.Ventil_UV02_GP02 := #In.Anf_HF_Ents_CM0x AND #In."SRM_GP02.QM41_auf" AND #In.Auto
               AND #In.Tuer_zu_vorn_GP02 AND #Leckage_Entsorgung_ok_GP02;

               // Check Weg Verwerfen
               #Zst.Weg_frei := #In.SRM_Saugseite_auf AND
               (#In.SRM_UV02_GP01_auf AND #In.SRM_UV02_GP02_zu OR
               #In.SRM_UV02_GP02_auf AND #In.SRM_UV02_GP01_zu);

               #Out.Entsorgung_UV02 := #In.Anf_HF_Ents_CM0x AND #Zst.Weg_frei AND NOT #Mld.UeW_Dfl_Ents;

               // Wenn geöffnet --> Frg Pumpe
               #Zst.Umwaelzen := (#In.SRM_Druckseite_auf AND  #In.SRM_Saugseite_auf) OR  (#Zst.Weg_frei AND #In.SRM_Entsogung_UV02_auf) ;

           1:  // Entsorgung --> GP02
                         // Ventile öffnen
               #Out.Ventil_Saugseite := #In.Ein AND #In.Niv_TLS AND #In.SRM_Ausgang_Spülltg_zu AND #In.SRM_Eingang_Spülltg_zu;
               #Out.Ventil_Druckseite := FALSE;

               // Verwerfen 
               #Out.Ventil_UV02_GP02 := #In.Ein AND #In."SRM_GP02.QM41_auf" AND #In.Tuer_zu_vorn_GP02
               AND #Leckage_Entsorgung_ok_GP02;

               // Check Weg Verwerfen
               #Zst.Weg_frei := #In.SRM_Saugseite_auf AND #In.SRM_UV02_GP02_auf AND #In.SRM_UV02_GP01_zu;

               #Out.Entsorgung_UV02 := #In.Ein AND #Zst.Weg_frei;

               // Wenn geöffnet --> Frg Pumpe
               #Zst.Umwaelzen := #Zst.Weg_frei AND #In.SRM_Entsogung_UV02_auf;

           2:  // Entsorgung --> GP01
                        // Ventile öffnen
               #Out.Ventil_Saugseite := #In.Ein AND #In.Niv_TLS AND #In.SRM_Ausgang_Spülltg_zu AND #In.SRM_Eingang_Spülltg_zu;
               #Out.Ventil_Druckseite := FALSE;

               // Verwerfen 
               #Out.Ventil_UV02_GP01 := #In.Ein AND #In."SRM_GP01.QM14_auf" AND #In.Tuer_zu_Seite_GP01 AND #In.Tuer_zu_vorn_GP01
               AND #Leckage_Entsorgung_ok_GP01;

               // Check Weg Verwerfen
               #Zst.Weg_frei := #In.SRM_Saugseite_auf AND #In.SRM_UV02_GP01_auf AND #In.SRM_UV02_GP02_zu;

               #Out.Entsorgung_UV02 := #In.Ein AND #Zst.Weg_frei;

               // Wenn geöffnet --> Frg Pumpe
               #Zst.Umwaelzen := #Zst.Weg_frei AND #In.SRM_Entsogung_UV02_auf;

           3: // Spülen - nur Hand
               #Zst.Umwaelzen := FALSE;
               #Zst.Weg_frei := FALSE;

               IF #In.Ein AND #In.Frg_Niv_CM05 THEN
                       IF #posFl_Hand THEN
                           #Zst.Spuelen_aktiv := TRUE;
                       END_IF;
                       #Out.Spülventil_Eingang := #In.SRM_Druckseite_zu AND #In.SRM_Saugseite_zu AND #Zst.Spuelen_aktiv;

                       #IEC_Timer.Spülen(IN := #In.SRM_Eingang_Spülltg_auf AND #In.SRM_Ausgang_Spülltg_auf,
                                         PT := #Param.Spülzeit,
                                         Q => #Zst.Spuelen,
                                         ET => #Spülzeit);
                       #Zst.Restzeit_Spülen := #Param.Spülzeit - #Spülzeit;

                       IF #In.SRM_Eingang_Spülltg_auf AND #In.SRM_Ausgang_Spülltg_auf AND NOT #Zst.Spuelen THEN
                           #Zst.Spuelen_aktiv := FALSE;
                           #Out.Spülventil_Eingang := FALSE;
                       END_IF;

                       // Fertig
                       IF NOT #Zst.Spuelen AND NOT #Zst.Spuelen_aktiv AND NOT #Out.Spülventil_Ausgang THEN
                           #Out.Spülventil_Eingang := FALSE;
                           #Out.Spülventil_Ausgang := FALSE;
                           #Zst.Restzeit_Spülen := T#0s;
                           #Mld.Pu_Spuelen_Fertig := TRUE;
                       END_IF;
                   ELSE
                       #Zst.Spuelen := FALSE;
                       #Out.Spülventil_Eingang := FALSE;
                       #Out.Spülventil_Ausgang := FALSE;
                       #Zst.Restzeit_Spülen := T#0s;
                   END_IF;

           4: // Spülen + Drucktest - nur Hand
               #Zst.Umwaelzen := FALSE;
               #Zst.Weg_frei := FALSE;
            IF NOT #Zst.Drucktest_aktiv THEN
                   IF #In.Ein AND #In.Frg_Niv_CM05 THEN
                       IF #posFl_Hand THEN
                           #Zst.Spuelen_aktiv := TRUE;
                       END_IF;
                       #Out.Spülventil_Eingang := #In.SRM_Druckseite_zu AND #In.SRM_Saugseite_zu;
                       #Out.Spülventil_Ausgang := #Out.Spülventil_Eingang;

                       #IEC_Timer.Spülen(IN := #In.SRM_Eingang_Spülltg_auf AND #In.SRM_Ausgang_Spülltg_auf,
                                         PT := #Param.Spülzeit,
                                         Q => #Zst.Spuelen,
                                         ET => #Spülzeit);
                       #Zst.Restzeit_Spülen := #Param.Spülzeit - #Spülzeit;

                       IF #In.SRM_Eingang_Spülltg_auf AND #In.SRM_Ausgang_Spülltg_auf AND NOT #Zst.Spuelen THEN
                           #Zst.Spuelen_aktiv := FALSE;
                       END_IF;

                       // Fertig
                       IF NOT #Zst.Spuelen AND NOT #Zst.Spuelen_aktiv THEN
                           #Out.Spülventil_Eingang := FALSE;
                           #Out.Spülventil_Ausgang := FALSE;
                           #Zst.Restzeit_Spülen := T#0s;
                            #Zst.Drucktest_aktiv := TRUE;
                            #Zst.Status_DT := #S1;
                       END_IF;
                   ELSE
                       #Zst.Spuelen := FALSE;
                       #Out.Spülventil_Eingang := FALSE;
                       #Out.Spülventil_Ausgang := FALSE;
                       #Zst.Restzeit_Spülen := T#0s;
                   END_IF;
                END_IF;

                IF #Zst.Drucktest_aktiv THEN

                    CASE #Zst.Status_DT OF

                        #S1:  //Druckaufbau
                            IF "DB_Temporaer".Drucksensoren_deaktiviert THEN//20.01.22
                                #Zst.Drucktest_ok := TRUE;

                                "Ergebnis_DT"("Name" := #Param.Name,
                                              akt_Zeit := "Uhrzeit".aktDatum,
                                              ok := #Zst.Drucktest_ok,
                                              Fehler := NOT #Zst.Drucktest_ok);

                                #Mld.Drucktest_ok := #Zst.Drucktest_ok;
                                #Mld.DT_Fehler := NOT #Zst.Drucktest_ok;

                                #Zst.Status_DT := #S4;
                            ELSE

                                #Out.Spülventil_Eingang := #In.SRM_Druckseite_zu AND #In.SRM_Saugseite_zu;
                                #Out.Spülventil_Ausgang := FALSE;
                                IF (#In.Druck_Pumpe > #Param.SW_Drucktest + 0.25) OR #Mld.TO_Druckaufbau THEN
                                    #Out.Spülventil_Eingang := FALSE;
                                    #Zst.Status_DT := #S2;
                                END_IF;
                                #Zst.Restzeit_DT := #Param.DT_Druckaufbau - #IEC_Timer.TO_Druckaufbau.ET;
                            END_IF;

                        #S2: //Wartezeit
                           #IEC_Timer.Drucktest(IN := #In.SRM_Eingang_Spülltg_zu,
                                                PT := #Param.DT_Testzeit,
                                                Q => #Zst.Zeit_laeuft,
                                                ET => #Zeit_DT);
                           #Zst.Restzeit_DT := #Param.DT_Testzeit - #Zeit_DT;

                           IF NOT #Zst.Zeit_laeuft AND #In.SRM_Eingang_Spülltg_zu THEN
                               #Zst.Restzeit_DT := T#0s;
                               #Zst.Status_DT := #S3;
                           END_IF;

                       #S3:// Überprüfung
                           #Zst.Drucktest_ok := #In.Druck_Pumpe >= #Param.SW_Drucktest;

                           "Ergebnis_DT"("Name" := #Param.Name,
                                         akt_Zeit := "Uhrzeit".aktDatum,
                                         ok := #Zst.Drucktest_ok,
                                         Fehler := NOT #Zst.Drucktest_ok);

                           #Mld.Drucktest_ok := #Zst.Drucktest_ok;
                           #Mld.DT_Fehler := NOT #Zst.Drucktest_ok;

                           #Zst.Status_DT := #S4;

                       #S4: // Ende
                           ;
                   END_CASE;
               END_IF;
       END_CASE;
   END_IF;

       // Pumpe an    
   #Out.GP0x_Ein := (#Zst.Umwaelzen (*OR #Zst.Spuelen*)) AND NOT #In.NotHalt AND #In.ext_Freigabe;

       // Geschwindigkeitsvorgabe
       // SEW: 100% == 3000 U/min == 15000 Digits
       IF #Out.GP0x_Ein THEN
           IF #In.Ein THEN
               #Out.Soll_speed := #Param.SW_Hand * 150;
           ELSE
               IF "Uhrzeit".AZ_aktiv THEN
                   #Out.Soll_speed := #Param.SW_Auto_AZ * 150;
               ELSE
                   #Out.Soll_speed := #Param.SW_Auto_aAZ * 150;
               END_IF;
           END_IF;
       ELSE
           #Out.Soll_speed := 0;
       END_IF;
END_REGION

REGION Network 3 (SCL): Überwachung / Meldungen
   // Trockenlaufschutz
   #Mld.Niv_TLS := NOT #In.Niv_TLS;
   // Überlauf
   #Mld.Niv_Ueberlauf := #In.Niv_Uel;

   // Durchflussüberwachung
   #IEC_Timer.Imp_Dfl(IN := NOT #In.Imp_Dfl AND #Zst.Umwaelzen AND #Out.Entsorgung_UV02,
                      PT := T#5s,
                      Q => #Alarm_Dfl_Ents);

   IF #Alarm_Dfl_Ents THEN
       #Mld.UeW_Dfl_Ents := TRUE;
   END_IF;

   // Zeitüberschreitung Druckaufbau
   #IEC_Timer.TO_Druckaufbau(IN := #Zst.Status_DT = #S1,
                             PT := #Param.DT_Druckaufbau,
                             Q => #Mld.TO_Druckaufbau);

   // Grenzwert Druck
   #IEC_Timer.GW_p(IN :=#Out.GP0x_Ein AND #In.GW_p_UP,
                   PT := T#3s,
                   Q => #Mld.GW_p_UP);

   #IEC_Timer.GW_Dfl(IN := #In.GW_Dfl AND #Out.GP0x_Ein AND #In.SRM_Druckseite_auf AND #Out.Entsorgung_UV02,
                     PT := T#15s,
                     Q => #Mld.GW_Dfl);

   // Grenzwert Leitfähigkeit Düsen Umwälzung
   #Mld.GW_LF_UP := #In.GW_LF_UP;

   // Frequenzumrichter 24V-Betrieb
   #Mld.FU_nicht_bereit := NOT #In.FU_betriebsbereit AND NOT #In.NotHalt;
   // Störung Frequenzumrichter
   #Mld.FU_Stoerung := #In.FU_Stoerung AND NOT #In.NotHalt;
   // nicht in Automatik
   #Mld.n_Auto := NOT #In.Auto AND "DB_ANLAGE".BA.Automat_ein;
END_REGION

REGION Network 4 (SCL): --> Visu
   // Status Pumpe
   "Status_E0A"(Hand := #In.Ein,
                Auto := #In.Auto,
                SonderModus_PumpeSpuelen:=#Zst.Spuelen,
                Stoerung := #In.FU_Stoerung OR NOT #In.FU_betriebsbereit,
                Ausgang := #Out.GP0x_Ein,
                StatusByte => #Zst.Status_GP0x);

   // Ist-Geschwindigkeit FU
   // SEW: 100% == 3000 U/min == 15000 Digits
   #Zst.speed := #In.FU_speed / 150; // in[%]

   // Anzeige Füllstand
   "Niv_Visu"(Niv_1 := #In.Niv_TLS,
              Niv_2 := #In.Niv_min,
              Niv_3 := #In.Niv_max,
              Niv_4 := #In.Niv_Uel,
              Niv_5 := FALSE,
              Niv_6 := FALSE,
              Wert_1 := #Niv_TLS,
              Wert_2 := #Niv_Min,
              Wert_3 := #Niv_max,
              Wert_4 := #Niv_Uel,
              Wert_5 := 0,
              Wert_6 := 0,
              Niveau => #Zst.Niveau,
              Niv_Err => #Mld.Niv_Sensorfehler);
END_REGION
END_FUNCTION_BLOCK

FUNCTION_BLOCK "UP_Spuele.GP0x"   // FB1003, LAD
TITLE = Umwälzpumpe Spüle
{ S7_Optimized_Access := 'TRUE' }
// Funktionen:  Entleeren /  Spülen
// stored: AutoNumber false, MemoryReserve 100, SetENOAutomatically false
   VAR RETAIN
      In { ExternalAccessible := 'False'; ExternalVisible := 'False'; ExternalWritable := 'False'} : Struct
         NotHalt : Bool;
         ext_Freigabe : Bool;   // kein Gasalarm, Kein Notstrom
         TW_senkt : Bool;
         Auto : Bool;   // Paneltaste
         Ein : Bool;   // Paneltaste
         FU_betriebsbereit : Bool;
         FU_Stoerung : Bool;
         Niv_TLS : Bool;
         Niv_min : Bool;
         Frg_Niv_CM05 : Bool;
         SRM_Saugseite_auf : Bool;
         SRM_Saugseite_zu : Bool;
         SRM_Druckseite_auf : Bool;
         SRM_Druckseite_zu : Bool;
         GW_p_UP : Bool;
         Betriebsart : USInt := 0;   // Paneltaste
         FU_speed : Int;
         Druck_Pumpe : Real;
      END_STRUCT;
      Param { ExternalAccessible := 'False'; ExternalVisible := 'False'; ExternalWritable := 'False'} : Struct
         SW_Hand : Int;   // [%]
         SW_Auto_AZ : Int;   // [%]
         SW_Auto_aAZ : Int;   // [%]
         Spülzeit : Time;
         DT_Druckaufbau : Time;
         DT_Testzeit : Time;
         SW_Drucktest : Real;
         "Name" : String[12];
      END_STRUCT;
      Zst { ExternalAccessible := 'False'; ExternalVisible := 'False'; ExternalWritable := 'False'} : Struct
         Niveau : USInt;
         Status_GP0x : USInt;
         Status_DT : USInt;
         Restzeit_Spülen : Time;
         Restzeit_DT : Time;
         TON_Spülventil_auf : Bool;
         Spuelen : Bool;
         Spuelen_aktiv : Bool;
         Drucktest_aktiv : Bool;
         Umwaelzen : Bool;
         Zeit_laeuft : Bool;
         Drucktest_ok : Bool;
         Bedienung_erlaubt : Bool;
         speed : Int;   // [%]
      END_STRUCT;
      Mld { ExternalAccessible := 'False'; ExternalVisible := 'False'; ExternalWritable := 'False'} : Struct
         Niv_TLS : Bool;
         Niv_Sensorfehler : Bool;
         GW_p_UP : Bool;
         FU_nicht_bereit : Bool;
         FU_Stoerung : Bool;
         n_Auto : Bool;
         TO_Druckaufbau : Bool;
         Drucktest_ok : Bool;
         DT_Fehler : Bool;
         Pu_Spuelen_Fertig : Bool;
      END_STRUCT;
      Out { ExternalAccessible := 'False'; ExternalVisible := 'False'; ExternalWritable := 'False'} : Struct
         GP0x_Ein : Bool;
         Ventil_Saugseite : Bool;
         Ventil_Druckseite : Bool;
         Spülventil : Bool;
         Ventil_CM05 : Bool;
         Soll_speed : Int;
      END_STRUCT;
   END_VAR
   VAR
      IEC_Timer { ExternalAccessible := 'False'; ExternalVisible := 'False'; ExternalWritable := 'False'} : Struct
         Spülventil_auf { S7_SetPoint := 'True'} : TON_TIME;
         Spülen { S7_SetPoint := 'True'} : TP_TIME;
         GW_p { S7_SetPoint := 'True'} : TON_TIME;
         Drucktest { S7_SetPoint := 'True'} : TP_TIME;
         TO_Druckaufbau { S7_SetPoint := 'True'} : TON_TIME;
         Ventil_CMO5 { S7_SetPoint := 'True'} : TOF_TIME;
      END_STRUCT;
      R_TRIG_Hand_EIN { ExternalAccessible := 'False'; ExternalVisible := 'False'; ExternalWritable := 'False'} : R_TRIG;
   END_VAR
   VAR_TEMP
      Spülzeit : Time;
      Zeit_DT : Time;
      posFl_Hand : Bool;
   END_VAR
   VAR CONSTANT
      Niv_TLS : USInt := 7;
      Niv_Min : USInt := 70;
      Niv_max : USInt := 85;
      Zeit_Ventil_auf : Time := T#1s;
      S1 : USInt := 1;
      S2 : USInt := 2;
      S3 : USInt := 3;
      S4 : USInt := 4;
   END_VAR
BEGIN

REGION Network 1 (SCL): Input
   // Panelbedienung und Sensoren --> Input()
   // Not-Halt
   #In.NotHalt := NOT "DB_PNOZ_IN_Out".In.NH_Frg_Pumpen OR NOT "E_Frg_AbLW";

   // Timer Spülventil AUF
   #IEC_Timer.Spülventil_auf(IN := #Out.Spülventil,
                              PT := #Zeit_Ventil_auf,
                              Q => #Zst.TON_Spülventil_auf);

    // positive Flanke "Hand Ein"
   #R_TRIG_Hand_EIN(CLK := #In.Ein,
                    Q => #posFl_Hand);
END_REGION

REGION Network 2 (SCL): Ansteuerung

   // "Normal"-Betrieb
   #Zst.Bedienung_erlaubt := NOT #In.Ein AND NOT #In.Auto AND NOT #Mld.DT_Fehler;

   //Drucktest rücksetzen
   IF #In.Betriebsart <> 2 OR #Zst.Spuelen_aktiv OR #Zst.Umwaelzen OR NOT #In.Ein THEN
       #Mld.Drucktest_ok := FALSE;
       // #Mld.DT_Fehler := FALSE;
       #Mld.TO_Druckaufbau := FALSE;
       #Zst.Status_DT := 0;
       #Zst.Drucktest_aktiv := FALSE;
   END_IF;
   //Spülmeldung rücksetzen
   IF #In.Betriebsart <> 1 OR NOT #In.Ein THEN
       #Mld.Pu_Spuelen_Fertig := FALSE;
   END_IF;

       CASE #In.Betriebsart OF
           0:  // Umwälzen

               // Spülventil zu
               #Out.Spülventil := FALSE;
               #Out.Ventil_CM05 := FALSE;
               #Zst.Restzeit_Spülen := T#0s;
               // Ventile öffnen
               #Out.Ventil_Saugseite := (#In.Auto OR #In.Ein) AND #In.Niv_TLS AND NOT #In.TW_senkt;
               #Out.Ventil_Druckseite := #Out.Ventil_Saugseite;
               // Wenn geöffnet --> Frg Pumpe
               #Zst.Umwaelzen := #In.SRM_Druckseite_auf AND #In.SRM_Saugseite_auf;
               #Zst.Drucktest_aktiv := FALSE;

           1: // Spülen - nur Hand
               #Zst.Umwaelzen := FALSE;
               #Out.Ventil_Saugseite := FALSE;
               #Out.Ventil_Druckseite := FALSE;

               // Ausschaltverzögert - Druckabbau
               #IEC_Timer.Ventil_CMO5(IN := #Out.Spülventil,
                                      PT := T#3s,
                                      Q => #Out.Ventil_CM05);

                   IF #In.Ein AND #In.Frg_Niv_CM05 THEN
                       IF #posFl_Hand THEN
                           #Zst.Spuelen_aktiv := TRUE;
                       END_IF;

                       #Out.Spülventil := #In.SRM_Druckseite_zu AND #In.SRM_Saugseite_zu AND #Zst.Spuelen_aktiv;

                       #IEC_Timer.Spülen(IN := #Zst.TON_Spülventil_auf,
                                         PT := #Param.Spülzeit,
                                         Q => #Zst.Spuelen,
                                         ET => #Spülzeit);
                       #Zst.Restzeit_Spülen := #Param.Spülzeit - #Spülzeit;

                       IF #Zst.TON_Spülventil_auf AND #In.SRM_Saugseite_zu AND #In.SRM_Druckseite_zu
                           AND NOT #Zst.Spuelen AND #Zst.Spuelen_aktiv THEN
                           #Zst.Spuelen_aktiv := FALSE;
                           #Out.Spülventil := FALSE;
                       END_IF;

                       // Fertig
                       IF NOT #Zst.Spuelen AND NOT #Zst.Spuelen_aktiv AND NOT #Out.Ventil_CM05 THEN
                           #Out.Spülventil := FALSE;
                           #Out.Ventil_CM05 := FALSE;
                           #Zst.Restzeit_Spülen := T#0s;
                           #Mld.Pu_Spuelen_Fertig := TRUE;
                       END_IF;
                   ELSE
                       #Zst.Spuelen := FALSE;
                       #Out.Spülventil := FALSE;
                       #Out.Ventil_CM05 := FALSE;
                       #Zst.Restzeit_Spülen := T#0s;
                   END_IF;

           2: // Spülen + Drucktest - nur Hand
               #Zst.Umwaelzen := FALSE;
               #Out.Ventil_Saugseite := FALSE;
               #Out.Ventil_Druckseite := FALSE;
               IF NOT #Zst.Drucktest_aktiv THEN
                   IF #In.Ein AND #In.Frg_Niv_CM05 THEN
                       IF #posFl_Hand THEN
                           #Zst.Spuelen_aktiv := TRUE;
                       END_IF;

                       #Out.Spülventil := #In.SRM_Druckseite_zu AND #In.SRM_Saugseite_zu AND #Zst.Spuelen_aktiv;
                       #Out.Ventil_CM05 := #Out.Spülventil;

                       #IEC_Timer.Spülen(IN := #Zst.TON_Spülventil_auf,
                                         PT := #Param.Spülzeit,
                                         Q => #Zst.Spuelen,
                                         ET => #Spülzeit);
                       IF #Zst.TON_Spülventil_auf AND #In.SRM_Saugseite_zu AND #In.SRM_Druckseite_zu
                           AND NOT #Zst.Spuelen AND #Zst.Spuelen_aktiv THEN
                           #Zst.Spuelen_aktiv := FALSE;
                       END_IF;
                       #Zst.Restzeit_Spülen := #Param.Spülzeit - #Spülzeit;
                       // Fertig
                       IF NOT #Zst.Spuelen AND NOT #Zst.Spuelen_aktiv THEN
                           #Out.Spülventil := FALSE;
                           #Out.Ventil_CM05 := FALSE;
                           #Zst.Restzeit_Spülen := T#0s;
                           #Zst.Drucktest_aktiv := TRUE;
                           #Zst.Status_DT := #S1;
                       END_IF;
                   ELSE
                       #Zst.Spuelen := FALSE;
                       #Out.Spülventil := FALSE;
                       #Out.Ventil_CM05 := FALSE;
                       #Zst.Restzeit_Spülen := T#0s;
                   END_IF;
               END_IF;

               IF #Zst.Drucktest_aktiv THEN
                   CASE #Zst.Status_DT OF
                       #S1:  //Druckaufbau
                           IF "DB_Temporaer".Drucksensoren_deaktiviert THEN//20.01.22
                               #Zst.Drucktest_ok := TRUE;

                               "Ergebnis_DT"("Name" := #Param.Name,
                                             akt_Zeit := "Uhrzeit".aktDatum,
                                             ok := #Zst.Drucktest_ok,
                                             Fehler := NOT #Zst.Drucktest_ok);

                               #Mld.Drucktest_ok := #Zst.Drucktest_ok;
                               #Mld.DT_Fehler := NOT #Zst.Drucktest_ok;
                               #Zst.Status_DT := #S4;
                           ELSE
                               #Out.Spülventil := #In.SRM_Druckseite_zu AND #In.SRM_Saugseite_zu;
                               #Out.Ventil_CM05 := FALSE;
                               IF (#In.Druck_Pumpe > #Param.SW_Drucktest + 0.25) OR #Mld.TO_Druckaufbau THEN
                                   #Zst.Status_DT := #S2;
                               END_IF;
                               #Zst.Restzeit_DT := #Param.DT_Druckaufbau - #IEC_Timer.TO_Druckaufbau.ET;
                           END_IF;
                       #S2: //Wartezeit
                           #IEC_Timer.Drucktest(IN := NOT #Out.Spülventil,
                                                PT := #Param.DT_Testzeit,
                                                Q => #Zst.Zeit_laeuft,
                                                ET => #Zeit_DT);
                           #Zst.Restzeit_DT := #Param.DT_Testzeit - #Zeit_DT;

                           IF NOT #Zst.Zeit_laeuft AND NOT #Out.Spülventil THEN
                               #Zst.Restzeit_DT := T#0s;
                               #Zst.Status_DT := #S3;
                           END_IF;
                           #Out.Spülventil := FALSE;
                           #Out.Ventil_CM05 := FALSE;
                       #S3:// Überprüfung
                           #Zst.Drucktest_ok := #In.Druck_Pumpe >= #Param.SW_Drucktest;

                           "Ergebnis_DT"("Name" := #Param.Name,
                                         akt_Zeit := "Uhrzeit".aktDatum,
                                         ok := #Zst.Drucktest_ok,
                                         Fehler := NOT #Zst.Drucktest_ok);

                           #Mld.Drucktest_ok := #Zst.Drucktest_ok;
                           #Mld.DT_Fehler := NOT #Zst.Drucktest_ok;
                           #Zst.Status_DT := #S4;
                       #S4: // Ende
                           ;

                   END_CASE;
               END_IF;
       END_CASE;

       // Pumpe an    
       #Out.GP0x_Ein := #Zst.Umwaelzen AND NOT #In.NotHalt AND #In.ext_Freigabe;

       // Geschwindigkeitsvorgabe
       // SEW: 100% == 3000 U/min == 15000 Digits
       IF #Out.GP0x_Ein THEN
           IF #In.Ein THEN
               #Out.Soll_speed := #Param.SW_Hand * 150;
           ELSE
               IF "Uhrzeit".AZ_aktiv THEN
                   #Out.Soll_speed := #Param.SW_Auto_AZ * 150;
               ELSE
                   #Out.Soll_speed := #Param.SW_Auto_aAZ * 150;
               END_IF;
           END_IF;
       ELSE
           #Out.Soll_speed := 0;
       END_IF;
END_REGION

REGION Network 3 (SCL): Überwachung / Meldungen
   // Trockenlaufschutz
   #Mld.Niv_TLS := NOT #In.Niv_TLS;

   // Zeitüberschreitung Druckaufbau
   #IEC_Timer.TO_Druckaufbau(IN := #Zst.Status_DT = #S1,
                             PT := #Param.DT_Druckaufbau,
                             Q => #Mld.TO_Druckaufbau);

   // Grenzwert Druck
   #IEC_Timer.GW_p(IN :=#Out.GP0x_Ein AND #In.GW_p_UP,
                   PT := T#3s,
                   Q => #Mld.GW_p_UP);
   // Frequenzumrichter 24V-Betrieb
   #Mld.FU_nicht_bereit := NOT #In.FU_betriebsbereit AND NOT #In.NotHalt;
   // Störung Frequenzumrichter
   #Mld.FU_Stoerung := #In.FU_Stoerung AND NOT #In.NotHalt;
   // nicht in Automatik
   #Mld.n_Auto := FALSE; //NOT #In.Auto AND "DB_ANLAGE".BA.Automat_ein;
END_REGION

REGION Network 4 (SCL): --> Visu
   // Status Pumpe
   "Status_E0A"(Hand := #In.Ein,
                Auto := #In.Auto,
                SonderModus_PumpeSpuelen:=#Zst.Spuelen,
                Stoerung := #In.FU_Stoerung OR NOT #In.FU_betriebsbereit,
                Ausgang := #Out.GP0x_Ein,
                StatusByte => #Zst.Status_GP0x);

   // Ist-Geschwindigkeit FU
   // SEW: 100% == 3000 U/min == 15000 Digits
   #Zst.speed := #In.FU_speed / 150; // in[%]

   // Anzeige Füllstand
   "Niv_Visu"(Niv_1 := #In.Niv_TLS,
              Niv_2 := #In.Niv_min,
              Niv_3 := FALSE,
              Niv_4 := FALSE,
              Niv_5 := FALSE,
              Niv_6 := FALSE,
              Wert_1 := #Niv_TLS,
              Wert_2 := #Niv_max,
              Wert_3 := 0,
              Wert_4 := 0,
              Wert_5 := 0,
              Wert_6 := 0,
              Niveau => #Zst.Niveau,
              Niv_Err => #Mld.Niv_Sensorfehler);
END_REGION
END_FUNCTION_BLOCK

FUNCTION_BLOCK "Pu_Versorgung.GP0x"   // FB1010, LAD
{ S7_Optimized_Access := 'TRUE' }
// Funktionen:  HF Versorgung  / Spülen
// stored: AutoNumber false, MemoryReserve 100, SetENOAutomatically false
   VAR RETAIN
      In { ExternalVisible := 'False'; ExternalWritable := 'False'} : Struct
         Auto : Bool;   // Paneltaste
         Ein : Bool;   // Paneltaste
         Not_Halt : Bool;
         Quitt_Al_Dfl : Bool;
         kein_Gas_Alarm : Bool;
         Leckage_Pumpe_ok : Bool;
         Leckage_PFA_Uebergang_ok : Bool;
         Leckage_Doppelrohr_ok : Bool;
         Leckage_Uml_Tunnel_ok : Bool;
         Leckage_Doppelschlauch_ok : Bool;
         Niv_min : Bool;
         Niv_max : Bool;
         Niv_Min_CM01 : Bool;
         Niv_Max_CM01 : Bool;
         Niv_Übervoll_CM01 : Bool;
         Niv_Min_CM02 : Bool;
         Niv_Max_CM02 : Bool;
         Niv_Übervoll_CM02 : Bool;
         Frg_Niv_CM05 : Bool;
         SRM_Saugseite_auf : Bool;
         SRM_Saugseite_zu : Bool;
         SRM_Druckseite_auf : Bool;
         SRM_Druckseite_zu : Bool;
         SRM_Eingang_Spülltg_auf : Bool;
         SRM_Eingang_Spülltg_zu : Bool;
         SRM_Ausgang_Spülltg_auf : Bool;
         SRM_Ausgang_Spülltg_zu : Bool;
         SRM_Versogung_UV01_auf : Bool;
         SRM_Versogung_UV01_zu : Bool;
         SRM_UV01_CM01_auf : Bool;
         SRM_UV01_CM01_zu { ExternalAccessible := 'False'} : Bool;
         SRM_UV01_CM02_auf { ExternalAccessible := 'False'} : Bool;
         SRM_UV01_CM02_zu { ExternalAccessible := 'False'} : Bool;
         Anf_HF_CM01 { ExternalAccessible := 'False'} : Bool;
         Anf_HF_CM02 { ExternalAccessible := 'False'} : Bool;
         IBC_vorhanden { ExternalAccessible := 'False'} : Bool;
         Tuer_vorn_zu { ExternalAccessible := 'False'} : Bool;
         Tuer_seitlich_zu { ExternalAccessible := 'False'} : Bool;
         Imp_Dfl { ExternalAccessible := 'False'} : Bool;
         GW_Dfl { ExternalAccessible := 'False'} : Bool;
         Betriebsart { ExternalAccessible := 'False'} : USInt := 0;   // Paneltaste
         Niveau { ExternalAccessible := 'False'} : USInt;
         Dfl { ExternalAccessible := 'False'} : Real;
      END_STRUCT;
      Param { ExternalAccessible := 'False'; ExternalVisible := 'False'; ExternalWritable := 'False'} : Struct
         Spülzeit : Time;
      END_STRUCT;
      Zst { ExternalAccessible := 'False'; ExternalVisible := 'False'; ExternalWritable := 'False'} : Struct
         Niveau : USInt;
         Status_GP0x : USInt;
         Restzeit_Spülen : Time;
         Spuelen : Bool;
         Pumpen : Bool;
         Weg_frei : Bool;
         Spuelen_aktiv : Bool;
         Bedienung_erlaubt : Bool;
      END_STRUCT;
      Mld { ExternalVisible := 'False'; ExternalWritable := 'False'} : Struct
         Leckage_Pumpe : Bool;
         Leckage_PFA_Uebergang : Bool;
         Leckage_Doppelrohr : Bool;
         Leckage_Uml_Tunnel : Bool;
         Leckage_Doppelschlauch : Bool;
         Niv_Sensorfehler : Bool;
         GW_Dfl : Bool;
         UeW_Dfl_Dos : Bool;
         Leermeldung : Bool;
         Vollmeldung : Bool;
         n_Auto : Bool;
         Radarsonde_niO : Bool;
      END_STRUCT;
      Out { ExternalVisible := 'False'; ExternalWritable := 'False'} : Struct
         GP0x_Ein : Bool;
         Spülventil_Eingang : Bool;
         Spülventil_Ausgang : Bool;
         Ventil_Saugseite : Bool;
         Ventil_Druckseite : Bool;
         Ventil_Entsorgung : Bool;
         Versorgung_UV01 : Bool;
         UV01_CM01 : Bool;
         UV01_CM02 : Bool;
      END_STRUCT;
   END_VAR
   VAR
      IEC_Timer : Struct
         GW_Dfl { ExternalAccessible := 'False'; ExternalVisible := 'False'; ExternalWritable := 'False'; S7_SetPoint := 'True'} : TON_TIME;
         Spülen { S7_SetPoint := 'True'} : TP_TIME;
         Verz_Min { S7_SetPoint := 'True'} : TON_TIME;
         Imp_Dfl { S7_SetPoint := 'True'} : TON_TIME;
         Spülventil_Ausgang { S7_SetPoint := 'True'} : TOF_TIME;
         Verz_NivMax { S7_SetPoint := 'True'} : TON_TIME;
      END_STRUCT;
      R_TRIG_Hand_EIN { S7_SetPoint := 'True'} : R_TRIG;
   END_VAR
   VAR_TEMP
      Spülzeit : Time;
      posFl_Hand : Bool;
      Leckage_Versorgung_ok : Bool;
      Alarm_Dfl_Dos : Bool;
   END_VAR
   VAR CONSTANT
      Niv_TLS : USInt := 2;
      Niv_Min : USInt := 20;
      Niv_max : USInt := 90;
      Zeit_Ventil_auf : Time := T#5s;
   END_VAR
BEGIN

REGION Network 1 (SCL): Input
   // Panelbedienung und Sensoren --> Input()

   // positive Flanke "Hand Ein"
   #R_TRIG_Hand_EIN(CLK := #In.Ein,
                    Q => #posFl_Hand);
   // Freigabe Not-Halt Pumpen
   #In.Not_Halt := NOT "DB_PNOZ_IN_Out".In.NH_Frg_Pumpen OR NOT "E_Frg_AbLW";

   // Leckage Versorgung
   #Leckage_Versorgung_ok := #In.Leckage_Doppelrohr_ok AND #In.Leckage_PFA_Uebergang_ok AND #In.Leckage_Uml_Tunnel_ok AND #In.Leckage_Doppelschlauch_ok;

   // Quittierung Alarm Durchfluss
   IF #In.Quitt_Al_Dfl AND #Mld.UeW_Dfl_Dos THEN
       #Mld.UeW_Dfl_Dos := FALSE;
   END_IF;
END_REGION

REGION Network 2 (SCL): Ansteuerung
   // Alles AUS
   IF (#In.Betriebsart = 3) AND #In.Tuer_vorn_zu AND #In.Tuer_seitlich_zu AND NOT #In.Not_Halt THEN // Spülen
       // Ausschaltverzögert - Druckabbau
       #IEC_Timer.Spülventil_Ausgang(IN := #Out.Spülventil_Eingang,
                                     PT := T#3s,
                                     Q => #Out.Spülventil_Ausgang);
   ELSE
       #Out.Spülventil_Eingang := FALSE;
       #Out.Spülventil_Ausgang := FALSE;
   END_IF;

   #Zst.Restzeit_Spülen := T#0s;
   #Out.Ventil_Saugseite := FALSE;
   #Out.Ventil_Druckseite := FALSE;
   #Out.Versorgung_UV01 := FALSE;
   #Out.UV01_CM01 := FALSE;
   #Out.UV01_CM02 := FALSE;
   #Out.Ventil_Entsorgung := FALSE;
   #Out.GP0x_Ein := FALSE;

   IF #In.Tuer_vorn_zu AND #In.Tuer_seitlich_zu AND NOT #In.Not_Halt THEN
       CASE #In.Betriebsart OF
           0:  // Versorgung Auto

               // Ventile öffnen
               IF #Leckage_Versorgung_ok AND #In.kein_Gas_Alarm THEN
                   #Out.Ventil_Saugseite := #Out.Ventil_Druckseite := #Out.Versorgung_UV01 := #In.Auto;
                   #Out.UV01_CM01 := #In.Anf_HF_CM01 AND #In.Auto;
                   #Out.UV01_CM02 := #In.Anf_HF_CM02 AND #In.Auto;
               END_IF;

               // Check weg
               #Zst.Weg_frei := #In.SRM_Ausgang_Spülltg_zu AND #In.SRM_Eingang_Spülltg_zu AND
               #In.SRM_Druckseite_auf AND #In.SRM_Saugseite_auf AND #In.SRM_Versogung_UV01_auf AND
               ((#In.SRM_UV01_CM01_auf AND #In.SRM_UV01_CM02_zu AND #In.Anf_HF_CM01) OR (#In.SRM_UV01_CM02_auf AND #In.SRM_UV01_CM01_zu AND #In.Anf_HF_CM02));

               // Weg frei, Behälter nicht leer und Ziel nicht übervoll
               #Zst.Pumpen := #Zst.Weg_frei AND NOT #Mld.Leermeldung AND #In.IBC_vorhanden AND NOT #Mld.UeW_Dfl_Dos AND
               ((#In.Anf_HF_CM01 AND NOT #In.Niv_Übervoll_CM01 AND NOT #In.Niv_Max_CM01) OR (#In.Anf_HF_CM02 AND NOT #In.Niv_Übervoll_CM02 AND NOT #In.Niv_Max_CM02));

           1:  // Versorgung CM01 Hand
               // Ventile öffnen
               IF #Leckage_Versorgung_ok AND #In.kein_Gas_Alarm THEN
                   #Out.Ventil_Saugseite := #Out.Ventil_Druckseite := #Out.Versorgung_UV01 := #Out.UV01_CM01 := #In.Ein;
               END_IF;

               // Check weg
               #Zst.Weg_frei := #In.SRM_Ausgang_Spülltg_zu AND #In.SRM_Eingang_Spülltg_zu AND
               #In.SRM_Druckseite_auf AND #In.SRM_Saugseite_auf AND
               #In.SRM_Versogung_UV01_auf AND #In.SRM_UV01_CM01_auf AND #In.SRM_UV01_CM02_zu;

               // Weg frei, Behälter nicht leer und Ziel nicht übervoll
               #Zst.Pumpen := #Zst.Weg_frei AND NOT #Mld.Leermeldung AND #In.IBC_vorhanden AND NOT #In.Niv_Übervoll_CM01 AND NOT #In.Niv_Max_CM01 AND NOT #In.Niv_Min_CM01;

           2:  // Versorgung CM02 Hand
               // Ventile öffnen
               IF #Leckage_Versorgung_ok AND #In.kein_Gas_Alarm THEN
                   #Out.Ventil_Saugseite := #Out.Ventil_Druckseite := #Out.Versorgung_UV01 := #Out.UV01_CM02 := #In.Ein;
               END_IF;

               // Check Weg
               #Zst.Weg_frei := #In.SRM_Ausgang_Spülltg_zu AND #In.SRM_Eingang_Spülltg_zu AND
               #In.SRM_Druckseite_auf AND #In.SRM_Saugseite_auf AND
               #In.SRM_Versogung_UV01_auf AND #In.SRM_UV01_CM02_auf AND #In.SRM_UV01_CM01_zu;

               // Weg frei, Behälter nicht leer und Ziel nicht übervoll
               #Zst.Pumpen := #Zst.Weg_frei AND NOT #Mld.Leermeldung AND #In.IBC_vorhanden AND NOT #In.Niv_Übervoll_CM02 AND NOT #In.Niv_Max_CM02 AND NOT #In.Niv_Min_CM02;

           3: // Spülen - nur Hand
               #Zst.Pumpen := FALSE;

               IF #In.Ein THEN
                   IF #posFl_Hand THEN
                       #Zst.Spuelen_aktiv := TRUE;
                   END_IF;
                   #Out.Spülventil_Eingang := #In.Frg_Niv_CM05 AND #In.SRM_Saugseite_zu AND #In.SRM_Druckseite_zu AND #Zst.Spuelen_aktiv;

                   #IEC_Timer.Spülen(IN := #In.SRM_Eingang_Spülltg_auf AND #In.SRM_Ausgang_Spülltg_auf,
                                     PT := #Param.Spülzeit,
                                     Q => #Zst.Spuelen,
                                     ET => #Spülzeit);
                   #Zst.Restzeit_Spülen := #Param.Spülzeit - #Spülzeit;

                   IF #In.SRM_Eingang_Spülltg_auf AND #In.SRM_Ausgang_Spülltg_auf AND #In.SRM_Saugseite_zu AND #In.SRM_Druckseite_zu
                       AND NOT #Zst.Spuelen AND #Zst.Spuelen_aktiv THEN
                       #Zst.Spuelen_aktiv := FALSE;
                       #Out.Spülventil_Eingang := FALSE;
                   END_IF;

               ELSE
                   #Out.Spülventil_Eingang := FALSE;
                   #Out.Spülventil_Ausgang := FALSE;
                   #Zst.Spuelen := FALSE;
                   #Zst.Spuelen_aktiv := FALSE;
               END_IF;

           4: // Entsorgung
               #Zst.Spuelen := FALSE;
               #Zst.Pumpen := FALSE;

               //Quick Connect Entsorgung
               #Out.Ventil_Entsorgung := NOT #In.Niv_max AND (#In.Niveau < 85) AND #In.IBC_vorhanden;

       END_CASE;
       // Pumpe an 
       #Out.GP0x_Ein := #Zst.Pumpen AND #In.Leckage_Pumpe_ok;
   END_IF;
END_REGION

REGION Network 3 (SCL): Überwachung / Meldungen
   // Durchflussüberwachung
   #IEC_Timer.Imp_Dfl(IN := NOT #In.Imp_Dfl AND #Zst.Pumpen AND (#In.Anf_HF_CM01 OR #In.Anf_HF_CM02),
                       PT := T#5s,
                       Q => #Alarm_Dfl_Dos);

    IF #Alarm_Dfl_Dos THEN
        #Mld.UeW_Dfl_Dos := TRUE;
    END_IF;

   // Meldungen Leckage 

   #Mld.Leckage_Pumpe := NOT #In.Leckage_Pumpe_ok;

   #Mld.Leckage_PFA_Uebergang := NOT #In.Leckage_PFA_Uebergang_ok;

   #Mld.Leckage_Doppelrohr := NOT #In.Leckage_Doppelrohr_ok;

   #Mld.Leckage_Uml_Tunnel := NOT #In.Leckage_Uml_Tunnel_ok;

   #Mld.Leckage_Doppelschlauch := NOT #In.Leckage_Doppelschlauch_ok;

   #IEC_Timer.GW_Dfl(IN := #In.GW_Dfl AND #Out.GP0x_Ein AND #In.SRM_Druckseite_auf,
                     PT := T#5s,
                     Q => #Mld.GW_Dfl);

   // Verzögerung Leermeldung
   #IEC_Timer.Verz_Min(IN := NOT #In.Niv_min AND #In.SRM_Saugseite_auf,
                       PT := T#5s,
                       Q => #Mld.Leermeldung);

   #Mld.Vollmeldung := #In.Niv_max AND (#In.Betriebsart = 4) AND #In.IBC_vorhanden;

   // nicht in Automatik
   #Mld.n_Auto := NOT #In.Auto AND "DB_ANLAGE".BA.Automat_ein AND #In.IBC_vorhanden;

   //Plausibiltät Radarsonde
   #Mld.Radarsonde_niO := ((#In.Niv_max AND (#In.Niveau < 85)) OR (NOT #In.Niv_max AND (#In.Niveau > 95)))
   AND #In.IBC_vorhanden;
END_REGION

REGION Network 4 (SCL): --> Visu
   // Status Pumpe
   "Status_E0A"(Hand := #In.Ein,
                Auto := #In.Auto,
                SonderModus_PumpeSpuelen:=FALSE,
                Stoerung := FALSE,
                Ausgang := #Out.GP0x_Ein,
                StatusByte => #Zst.Status_GP0x);
   // Anzeige Füllstand
   "Niv_Visu"(Niv_1 := #In.Niv_min,
              Niv_2 := #In.Niv_max,
              Niv_3 := FALSE,
              Niv_4 := FALSE,
              Niv_5 := FALSE,
              Niv_6 := FALSE,
              Wert_1 := #Niv_Min,
              Wert_2 := #Niv_max,
              Wert_3 := 0,
              Wert_4 := 0,
              Wert_5 := 0,
              Wert_6 := 0,
              Niveau => #Zst.Niveau,
              Niv_Err => #Mld.Niv_Sensorfehler);

   // Radarsonde
   #Zst.Niveau := #In.Niveau;
   #Zst.Bedienung_erlaubt := NOT #In.Ein AND NOT #In.Auto;
END_REGION
END_FUNCTION_BLOCK

FUNCTION_BLOCK "Pu_Entl.GP0x"   // FB1009, LAD
TITLE = Pumpe Abpumpen Sump
{ S7_Optimized_Access := 'TRUE' }
// Funktionen:  Entleeren /  Spülen
// stored: AutoNumber false, MemoryReserve 100, SetENOAutomatically false
   VAR RETAIN
      In { ExternalAccessible := 'False'; ExternalVisible := 'False'; ExternalWritable := 'False'} : Struct
         Auto : Bool;   // Paneltaste
         Ein : Bool;   // Paneltaste
         Leckage_ok : Bool;
         Frg_Niv_CM05 : Bool;
         Betriebsart : USInt := 0;   // Paneltaste
      END_STRUCT;
      Param { ExternalAccessible := 'False'; ExternalVisible := 'False'; ExternalWritable := 'False'} : Struct
         Spülzeit : Time;
      END_STRUCT;
      Zst { ExternalAccessible := 'False'; ExternalVisible := 'False'; ExternalWritable := 'False'} : Struct
         Niveau : USInt;
         Status_GP0x : USInt;
         Restzeit_Spülen : Time;
         TON_Spülventil_auf : Bool;
         Spuelen : Bool;
         Abpumpen : Bool;
         Bedienung_Erlaubt : Bool;
      END_STRUCT;
      Mld { ExternalAccessible := 'False'; ExternalVisible := 'False'; ExternalWritable := 'False'} : Struct
         Leckage : Bool;
         Niv_Sensorfehler : Bool;
         n_Auto : Bool;
      END_STRUCT;
      Out { ExternalAccessible := 'False'; ExternalVisible := 'False'; ExternalWritable := 'False'} : Struct
         GP0x_Ein : Bool;
         Spülventil : Bool;
      END_STRUCT;
   END_VAR
   VAR
      IEC_Timer { ExternalAccessible := 'False'; ExternalVisible := 'False'; ExternalWritable := 'False'} : Struct
         Leckage_ok { S7_SetPoint := 'True'} : TON_TIME;
         Spülventil_auf { S7_SetPoint := 'True'} : TON_TIME;
         Spülen { S7_SetPoint := 'True'} : TP_TIME;
         Leckage_niO { S7_SetPoint := 'True'} : TON_TIME;
      END_STRUCT;
      R_TRIG_Hand_EIN { ExternalAccessible := 'False'; ExternalVisible := 'False'; ExternalWritable := 'False'} : R_TRIG;
   END_VAR
   VAR_TEMP
      Spülzeit : Time;
      Leckage_ok_verz : Bool;
      posFl_Hand : Bool;
   END_VAR
   VAR CONSTANT
      Niv_TLS : USInt := 2;
      Niv_Min : USInt := 2;
      Niv_max : USInt := 20;
      Zeit_Ventil_auf : Time := T#1s;
   END_VAR
BEGIN

REGION Network 1 (SCL): Input
   // Panelbedienung und Sensoren --> Input()
   // Leckage o.k. verzögert
   #IEC_Timer.Leckage_ok(IN := #In.Leckage_ok,
                         PT := T#120s,
                         Q => #Leckage_ok_verz);

   // Timer Spülventil AUF
   #IEC_Timer.Spülventil_auf(IN := #Out.Spülventil,
                              PT := #Zeit_Ventil_auf,
                              Q => #Zst.TON_Spülventil_auf);

    // positive Flanke "Hand Ein"
   #R_TRIG_Hand_EIN(CLK := #In.Ein,
                    Q => #posFl_Hand);

   #IEC_Timer.Spülen(IN := #posFl_Hand AND #In.Betriebsart = 1,
                     PT := #Param.Spülzeit,
                     Q => #Zst.Spuelen,
                     ET => #Spülzeit);
END_REGION

REGION Network 2 (SCL): Ansteuerung
   // Zielbehälter nicht voll
   IF #In.Frg_Niv_CM05 THEN
       CASE #In.Betriebsart OF
           0:  // Entleeren

               // Spülventil zu
               #Out.Spülventil := FALSE;
               #Zst.Restzeit_Spülen := T#0s;

               // Wenn Leckage oder einmalig per Hand
               IF #In.Auto AND NOT #In.Leckage_ok OR #posFl_Hand THEN
                   #Zst.Abpumpen := TRUE;
               ELSIF #Leckage_ok_verz THEN
                   #Zst.Abpumpen := FALSE;
               END_IF;

           1: // Spülen - nur Hand
               IF #In.Ein THEN
                   IF #posFl_Hand THEN
                       #Out.Spülventil := TRUE;
                   ELSIF NOT #Zst.Spuelen AND #Zst.TON_Spülventil_auf THEN
                       #Out.Spülventil := FALSE;
                   END_IF;
                   #Zst.Restzeit_Spülen := #Param.Spülzeit - #Spülzeit;
               ELSE
                   #Zst.Spuelen := FALSE;
                   #Out.Spülventil := FALSE;
                   #Zst.Restzeit_Spülen := T#0s;
               END_IF;

               // Wenn Leckage 
               IF #Leckage_ok_verz OR (NOT #In.Auto AND NOT #In.Ein) THEN
                   #Zst.Abpumpen := FALSE;
               ELSIF NOT #In.Leckage_ok THEN
                   #Zst.Abpumpen := TRUE;
               END_IF;
       END_CASE;

       // Pumpe an    
       #Out.GP0x_Ein := #Zst.Abpumpen AND (#In.Auto OR #In.Ein);
   ELSE
       #Out.Spülventil := FALSE;
       #Zst.Restzeit_Spülen := T#0s;
       #Out.GP0x_Ein := FALSE;
   END_IF;
END_REGION

REGION Network 3 (SCL): Überwachung / Meldungen

   // Meldung Leckage verzögert
   #IEC_Timer.Leckage_niO(IN := NOT #In.Leckage_ok,
                   PT := T#30s,
                   Q => #Mld.Leckage);

   // nicht in Automatik
   #Mld.n_Auto := NOT #In.Auto AND "DB_ANLAGE".BA.Automat_ein;
END_REGION

REGION Network 4 (SCL): --> Visu
   // Status Pumpe
   "Status_E0A"(Hand := #In.Ein,
                Auto := #In.Auto,
                SonderModus_PumpeSpuelen:=FALSE,
                Stoerung := FALSE,
                Ausgang := #Out.GP0x_Ein,
                StatusByte => #Zst.Status_GP0x);
   // Anzeige Füllstand
   "Niv_Visu"(Niv_1 := TRUE,
              Niv_2 := NOT #In.Leckage_ok,
              Niv_3 := FALSE,
              Niv_4 := FALSE,
              Niv_5 := FALSE,
              Niv_6 := FALSE,
              Wert_1 := #Niv_Min,
              Wert_2 := #Niv_max,
              Wert_3 := 0,
              Wert_4 := 0,
              Wert_5 := 0,
              Wert_6 := 0,
              Niveau => #Zst.Niveau,
              Niv_Err => #Mld.Niv_Sensorfehler);

   #Zst.Bedienung_Erlaubt := NOT #In.Ein AND NOT #In.Auto;
END_REGION
END_FUNCTION_BLOCK

FUNCTION_BLOCK "Pu_CM05.GP11"   // FB1011, LAD
TITLE = Pumpe GP11: Entleeren CM05
{ S7_Optimized_Access := 'TRUE' }
// Funktionen:  Entleeren /  Spülen
// stored: AutoNumber false, MemoryReserve 100, SetENOAutomatically false
   VAR RETAIN
      In { ExternalVisible := 'False'; ExternalWritable := 'False'} : Struct
         NotHalt : Bool;
         MSS_ok : Bool;
         Auto : Bool;   // Paneltaste
         Ein : Bool;   // Paneltaste
         GW_p : Bool;
         "Niv_Uel_CM05.BL05" : Bool;
         "Niv_max_CM05.BL01" : Bool;
         "Niv_min_CM05.BL02" : Bool;
         "Niv_TLS_CM05.BL03" : Bool;
         AWA_ok : Bool;
         Frg_AWA : Bool;
         "SRM_CM05.QM61_auf" : Bool;
         "SRM_CM05.QM61_zu" : Bool;
         "SRM_CM05.QM64_auf" : Bool;
         "SRM_CM05.QM64_zu" : Bool;
         Betriebsart : USInt := 0;   // Paneltaste
         Druck_Pumpe { ExternalAccessible := 'False'} : Real;
      END_STRUCT;
      Param { ExternalVisible := 'False'; ExternalWritable := 'False'} : Struct
         Spülzeit : Time;
         DT_Druckaufbau { ExternalAccessible := 'False'} : Time;
         DT_Testzeit { ExternalAccessible := 'False'} : Time;
         SW_Drucktest { ExternalAccessible := 'False'} : Real;
      END_STRUCT;
      Zst : Struct
         Niveau : USInt;
         Status_GP11 : USInt;
         Status_DT { ExternalAccessible := 'False'; ExternalVisible := 'False'; ExternalWritable := 'False'} : USInt;
         Restzeit_Spülen : Time;
         Restzeit_DT { ExternalAccessible := 'False'; ExternalVisible := 'False'; ExternalWritable := 'False'} : Time;
         "TON_CM05.QM62_auf" : Bool;
         Spuelen : Bool;
         Zeit_laeuft { ExternalAccessible := 'False'; ExternalVisible := 'False'; ExternalWritable := 'False'} : Bool;
         Spuelen_aktiv : Bool;
         Drucktest_aktiv : Bool;
         Drucktest_ok { ExternalAccessible := 'False'; ExternalVisible := 'False'; ExternalWritable := 'False'} : Bool;
         Bedienung_erlaubt { ExternalAccessible := 'False'; ExternalVisible := 'False'; ExternalWritable := 'False'} : Bool;
      END_STRUCT;
      Mld { ExternalVisible := 'False'; ExternalWritable := 'False'} : Struct
         MSS : Bool;
         "TLS_CM05.BL03" : Bool;
         "Uel_CM05.BL05" : Bool;
         AWA_niO : Bool;
         keine_Frg_AWA : Bool;
         Niv_Sensorfehler : Bool;
         GW_p : Bool;
         n_Auto : Bool;
         TO_Druckaufbau { ExternalAccessible := 'False'} : Bool;
         Drucktest_ok { ExternalAccessible := 'False'} : Bool;
         DT_Fehler { ExternalAccessible := 'False'} : Bool;
         Pu_Spuelen_Fertig { ExternalAccessible := 'False'} : Bool;
      END_STRUCT;
      Out { ExternalVisible := 'False'; ExternalWritable := 'False'} : Struct
         GP11_Ein : Bool;
         QM61 : Bool;
         QM62 : Bool;
         QM63 : Bool;
         QM64 : Bool;
      END_STRUCT;
   END_VAR
   VAR
      IEC_Timer : Struct
         "CM05.QM62_auf" { ExternalAccessible := 'False'; ExternalVisible := 'False'; ExternalWritable := 'False'; S7_SetPoint := 'True'} : TON_TIME;
         Spülen { S7_SetPoint := 'True'} : TP_TIME;
         GW_p { S7_SetPoint := 'True'} : TON_TIME;
         Drucktest { ExternalAccessible := 'False'; ExternalVisible := 'False'; ExternalWritable := 'False'; S7_SetPoint := 'True'} : TP_TIME;
         TO_Druckaufbau { ExternalAccessible := 'False'; ExternalVisible := 'False'; ExternalWritable := 'False'; S7_SetPoint := 'True'} : TON_TIME;
         QM63 { S7_SetPoint := 'True'} : TOF_TIME;
      END_STRUCT;
      R_TRIG_Hand_EIN { S7_SetPoint := 'True'} : R_TRIG;
   END_VAR
   VAR_TEMP
      Spülzeit : Time;
      Zeit_DT : Time;
      GP11_Laeuft : Bool;
      posFl_Hand : Bool;
   END_VAR
   VAR CONSTANT
      Niv_TLS : USInt := 7;
      Niv_Min : USInt := 35;
      Niv_max : USInt := 85;
      Niv_Uel : USInt := 98;
      Zeit_Ventil_auf : Time := T#3s;
      S1 : USInt := 1;
      S2 : USInt := 2;
      S3 : USInt := 3;
      S4 : USInt := 4;
      "Name" : String := 'Pu CM05.GP11';
   END_VAR
BEGIN

REGION Network 1 (SCL): Input
   // Panelbedienung und Sensoren --> Input()
   // Not-Halt
   #In.NotHalt := NOT "DB_PNOZ_IN_Out".In.NH_Frg_Pumpen;
   // Timer Spülventil AUF
   #IEC_Timer."CM05.QM62_auf"(IN := #Out.QM62,
                              PT := #Zeit_Ventil_auf,
                              Q => #Zst."TON_CM05.QM62_auf");
   // positive Flanke "Hand Ein"
   #R_TRIG_Hand_EIN(CLK := #In.Ein,
                    Q => #posFl_Hand);
END_REGION

REGION Network 2 (SCL): Pumpe Ein Entleerung Sammeltank CM05.GP11
   IF #In.MSS_ok AND NOT #In.NotHalt THEN

       // "Normal"-Betrieb
       #Zst.Bedienung_erlaubt := NOT #In.Ein AND NOT #In.Auto AND NOT #Mld.DT_Fehler;

       //Drucktest rücksetzen
       IF #In.Betriebsart <> 2 OR #Zst.Spuelen_aktiv OR NOT #In.Ein THEN
           #Mld.Drucktest_ok := FALSE;
           #Mld.DT_Fehler := FALSE;
           #Mld.TO_Druckaufbau := FALSE;
           #Zst.Status_DT := 0;
           #Zst.Drucktest_aktiv := FALSE;
       END_IF;
       //Spülmeldung rücksetzen
       IF #In.Betriebsart <> 1 OR NOT #In.Ein THEN
           #Mld.Pu_Spuelen_Fertig := FALSE;
       END_IF;

       CASE #In.Betriebsart OF
           0:  // Entleeren
               #Out.QM64 := #In.AWA_ok AND #In.Frg_AWA;
               // Spülventile zu
               #Out.QM62 := FALSE;
               #Out.QM63 := FALSE;
               #Zst.Restzeit_Spülen := T#0s;
               #Zst.Drucktest_aktiv := FAlSE;

               // Zwischen MAX und MIN entleeren oder einmalig per Hand
               IF (#In.Auto AND #In."Niv_max_CM05.BL01" OR #posFl_Hand ) AND #In."Niv_TLS_CM05.BL03"THEN
                   #Out.QM61 := TRUE;
               ELSIF NOT #In."Niv_TLS_CM05.BL03" OR NOT #In."Niv_min_CM05.BL02" OR (NOT #In.Auto AND NOT #In.Ein) THEN
                       #Out.QM61 := FALSE;
                END_IF;

               //Pumpe an, wenn Ventile geöffnet sind
                #Out.GP11_Ein := #In."SRM_CM05.QM61_auf" AND #In."SRM_CM05.QM64_auf" AND #In."Niv_TLS_CM05.BL03";

            1: // Spülen - nur Hand
                // Ventile Abpumpen zu    
                #Out.QM61 := FALSE;
                #Out.QM64 := FALSE;

                // Ausschaltverzögert - Druckabbau
                #IEC_Timer.QM63(IN := #Out.QM62,
                                PT := T#3s,
                                Q => #Out.QM63);

                IF #In.Ein THEN
                        IF #posFl_Hand THEN
                            #Zst.Spuelen_aktiv := TRUE;
                        END_IF;
                        #Out.QM62 := NOT #In."Niv_max_CM05.BL01" AND #In."SRM_CM05.QM61_zu" AND #In."SRM_CM05.QM64_zu" AND NOT #In."Niv_Uel_CM05.BL05" AND #Zst.Spuelen_aktiv;

